QRS_NEXT_CUT()
PTP {E1 28976.886,E2 28976.886}
PTP {X 0,Y 607.919,A -85,B 0,C 180,E1 28976.886,E2 28976.886,E3 0,E4 0,E5 0,E6 0}
QRS_SPEED_INIT()
LIN {X 0,Y 607.919,Z 855,A -85,B 0,C 180,E1 28976.886,E2 28976.886,E3 0,E4 0,E5 0,E6 0} C_VEL
LIN {X 0,Y 607.919,Z 792.512,A -85,B 0,C 180,E1 28976.886,E2 28976.886} C_VEL
LIN {X 0,Y 607.919,Z 784.1,A -85,B 0,C 180,E1 28976.886,E2 28976.886} C_VEL
LIN {X 0,Y 607.91,Z 782.124,A -85,B 0,C 180,E1 28976.726,E2 28976.726} C_VEL
LIN {X 0,Y 607.918,Z 778.216,A -85,B 0,C 180,E1 28974.999,E2 28974.999} C_VEL
LIN {X 0,Y 607.918,Z 772.634,A -85,B 0,C 180,E1 28973.294,E2 28973.294} C_VEL
LIN {X 0,Y 607.917,Z 765.18,A -85,B 0,C 180,E1 28971.583,E2 28971.583} C_VEL
LIN {X 0,Y 607.91,Z 756.203,A -85,B 0,C 180,E1 28969.959,E2 28969.959} C_VEL
LIN {X 0,Y 607.915,Z 745.767,A -85,B 0,C 180,E1 28968.424,E2 28968.424} C_VEL
LIN {X 0,Y 607.915,Z 733.893,A -85,B 0,C 180,E1 28966.978,E2 28966.978} C_VEL
LIN {X 0,Y 607.913,Z 720.544,A -85,B 0,C 180,E1 28965.62,E2 28965.62} C_VEL
LIN {X 0,Y 607.917,Z 705.535,A -85,B 0,C 180,E1 28964.351,E2 28964.351} C_VEL
LIN {X 0,Y 607.92,Z 689.426,A -85,B 0,C 180,E1 28963.228,E2 28963.228} C_VEL
LIN {X 0,Y 607.911,Z 672.944,A -85,B 0,C 180,E1 28962.285,E2 28962.285} C_VEL
LIN {X 0,Y 607.914,Z 655.674,A -85,B 0,C 180,E1 28961.492,E2 28961.492} C_VEL
LIN {X 0,Y 607.918,Z 638.216,A -85,B 0,C 180,E1 28960.87,E2 28960.87} C_VEL
LIN {X 0,Y 607.911,Z 619.855,A -85,B 0,C 180,E1 28960.395,E2 28960.395} C_VEL
LIN {X 0,Y 607.907,Z 600.729,A -85,B 0,C 180,E1 28960.082,E2 28960.082} C_VEL
LIN {X 0,Y 607.893,Z 403.798,A -85,B 0,C 180,E1 28957.622,E2 28957.622} C_VEL
LIN {X 0,Y 607.907,Z 366.363,A -85,B 0,C 180,E1 28954.552,E2 28954.552} C_VEL
LIN {X 0,Y 607.851,Z 351.079,A -85,B 0,C 180,E1 28953.244,E2 28953.244} C_VEL
LIN {X 0,Y 607.85,Z 351.077,A -85,B 0,C 180,E1 28949.996,E2 28949.996} C_VEL
LIN {X 0,Y 607.849,Z 351.076,A -85,B 0,C 180,E1 28947.199,E2 28947.199} C_VEL
LIN {X 0,Y 607.849,Z 351.077,A -85,B 0,C 180,E1 28943.922,E2 28943.922} C_VEL
LIN {X 0,Y 607.845,Z 351.076,A -85,B 0,C 180,E1 28941.192,E2 28941.192} C_VEL
LIN {X 0,Y 607.851,Z 351.077,A -85,B 0,C 180,E1 28937.89,E2 28937.89} C_VEL
LIN {X 0,Y 607.845,Z 351.076,A -85,B 0,C 180,E1 28935.116,E2 28935.116} C_VEL
LIN {X 0,Y 607.851,Z 351.077,A -85,B 0,C 180,E1 28931.828,E2 28931.828} C_VEL
LIN {X 0,Y 607.845,Z 351.076,A -85,B 0,C 180,E1 28929.051,E2 28929.051} C_VEL
LIN {X 0,Y 607.848,Z 351.077,A -85,B 0,C 180,E1 28925.729,E2 28925.729} C_VEL
LIN {X 0,Y 607.845,Z 351.076,A -85,B 0,C 180,E1 28922.974,E2 28922.974} C_VEL
LIN {X 0,Y 607.848,Z 351.077,A -85,B 0,C 180,E1 28919.678,E2 28919.678} C_VEL
LIN {X 0,Y 607.845,Z 351.076,A -85,B 0,C 180,E1 28916.895,E2 28916.895} C_VEL
LIN {X 0,Y 607.845,Z 351.077,A -85,B 0,C 180,E1 28913.561,E2 28913.561} C_VEL
LIN {X 0,Y 607.847,Z 351.076,A -85,B 0,C 180,E1 28910.812,E2 28910.812} C_VEL
LIN {X 0,Y 607.846,Z 351.077,A -85,B 0,C 180,E1 28907.519,E2 28907.519} C_VEL
LIN {X 0,Y 607.843,Z 351.076,A -85,B 0,C 180,E1 28904.772,E2 28904.772} C_VEL
LIN {X 0,Y 607.848,Z 351.077,A -85,B 0,C 180,E1 28901.481,E2 28901.481} C_VEL
LIN {X 0,Y 607.845,Z 351.076,A -85,B 0,C 180,E1 28898.704,E2 28898.704} C_VEL
LIN {X 0,Y 607.845,Z 351.077,A -85,B 0,C 180,E1 28895.38,E2 28895.38} C_VEL
LIN {X 0,Y 607.844,Z 351.076,A -85,B 0,C 180,E1 28892.64,E2 28892.64} C_VEL
LIN {X 0,Y 607.847,Z 351.077,A -85,B 0,C 180,E1 28889.34,E2 28889.34} C_VEL
LIN {X 0,Y 607.848,Z 351.076,A -85,B 0,C 180,E1 28886.511,E2 28886.511} C_VEL
LIN {X 0,Y 607.848,Z 351.077,A -85,B 0,C 180,E1 28883.293,E2 28883.293} C_VEL
LIN {X 0,Y 607.842,Z 351.076,A -85,B 0,C 180,E1 28880.532,E2 28880.532} C_VEL
LIN {X 0,Y 607.85,Z 351.077,A -85,B 0,C 180,E1 28877.266,E2 28877.266} C_VEL
LIN {X 0,Y 607.837,Z 351.076,A -85,B 0,C 180,E1 28874.545,E2 28874.545} C_VEL
LIN {X 0,Y 607.864,Z 351.077,A -85,B 0,C 180,E1 28871.343,E2 28871.343} C_VEL
LIN {X 0,Y 607.833,Z 351.077,A -85,B 0,C 180,E1 28868.581,E2 28868.581} C_VEL
LIN {X 0,Y 607.885,Z 351.077,A -85,B 0,C 180,E1 28865.448,E2 28865.448} C_VEL
LIN {X 0,Y 607.832,Z 351.077,A -85,B 0,C 180,E1 28862.575,E2 28862.575} C_VEL
LIN {X 0,Y 607.906,Z 351.077,A -85,B 0,C 180,E1 28859.526,E2 28859.526} C_VEL
LIN {X 0,Y 607.83,Z 351.077,A -85,B 0,C 180,E1 28856.56,E2 28856.56} C_VEL
LIN {X 0,Y 607.913,Z 351.078,A -85,B 0,C 180,E1 28853.541,E2 28853.541} C_VEL
LIN {X 0,Y 607.83,Z 351.077,A -85,B 0,C 180,E1 28850.583,E2 28850.583} C_VEL
LIN {X 0,Y 607.903,Z 351.077,A -85,B 0,C 180,E1 28847.596,E2 28847.596} C_VEL
LIN {X 0,Y 607.831,Z 351.077,A -85,B 0,C 180,E1 28844.58,E2 28844.58} C_VEL
LIN {X 0,Y 607.883,Z 351.077,A -85,B 0,C 180,E1 28841.69,E2 28841.69} C_VEL
LIN {X 0,Y 607.832,Z 351.077,A -85,B 0,C 180,E1 28838.568,E2 28838.568} C_VEL
LIN {X 0,Y 607.859,Z 351.077,A -85,B 0,C 180,E1 28835.813,E2 28835.813} C_VEL
LIN {X 0,Y 607.837,Z 351.077,A -85,B 0,C 180,E1 28832.625,E2 28832.625} C_VEL
LIN {X 0,Y 607.855,Z 351.077,A -85,B 0,C 180,E1 28829.786,E2 28829.786} C_VEL
LIN {X 0,Y 607.837,Z 351.08,A -85,B 0,C 180,E1 28826.579,E2 28826.579} C_VEL
LIN {X 0,Y 607.829,Z 351.304,A -85,B 0,C 180,E1 28826.333,E2 28826.333} C_VEL
LIN {X 0,Y 607.917,Z 379.245,A -85,B 0,C 180,E1 28823.352,E2 28823.352} C_VEL
LIN {X 0,Y 607.876,Z 408.984,A -85,B 0,C 180,E1 28820.258,E2 28820.258} C_VEL
LIN {X 0,Y 607.915,Z 440.675,A -85,B 0,C 180,E1 28817.024,E2 28817.024} C_VEL
LIN {X 0,Y 607.889,Z 472.368,A -85,B 0,C 180,E1 28813.847,E2 28813.847} C_VEL
LIN {X 0,Y 607.915,Z 480.891,A -85,B 0,C 180,E1 28813.01,E2 28813.01} C_VEL
LIN {X 0,Y 607.868,Z 591.977,A -85,B 0,C 180,E1 28811.673,E2 28811.673} C_VEL
LIN {X 0,Y 607.896,Z 607.193,A -85,B 0,C 180,E1 28811.312,E2 28811.312} C_VEL
LIN {X 0,Y 607.914,Z 622.026,A -85,B 0,C 180,E1 28810.759,E2 28810.759} C_VEL
LIN {X 0,Y 607.88,Z 635.112,A -85,B 0,C 180,E1 28810.089,E2 28810.089} C_VEL
LIN {X 0,Y 607.918,Z 647.311,A -85,B 0,C 180,E1 28809.276,E2 28809.276} C_VEL
LIN {X 0,Y 607.919,Z 658.998,A -85,B 0,C 180,E1 28808.274,E2 28808.274} C_VEL
LIN {X 0,Y 607.918,Z 668.983,A -85,B 0,C 180,E1 28807.181,E2 28807.181} C_VEL
LIN {X 0,Y 607.917,Z 677.168,A -85,B 0,C 180,E1 28806.042,E2 28806.042} C_VEL
LIN {X 0,Y 607.918,Z 684.395,A -85,B 0,C 180,E1 28804.717,E2 28804.717} C_VEL
LIN {X 0,Y 607.917,Z 689.553,A -85,B 0,C 180,E1 28803.395,E2 28803.395} C_VEL
LIN {X 0,Y 607.916,Z 692.97,A -85,B 0,C 180,E1 28802.074,E2 28802.074} C_VEL
LIN {X 0,Y 607.918,Z 694.754,A -85,B 0,C 180,E1 28800.66,E2 28800.66} C_VEL
LIN {X 0,Y 607.914,Z 694.751,A -85,B 0,C 180,E1 28799.246,E2 28799.246} C_VEL
LIN {X 0,Y 607.919,Z 692.961,A -85,B 0,C 180,E1 28797.832,E2 28797.832} C_VEL
LIN {X 0,Y 607.919,Z 689.239,A -85,B 0,C 180,E1 28796.417,E2 28796.417} C_VEL
LIN {X 0,Y 607.916,Z 683.914,A -85,B 0,C 180,E1 28795.094,E2 28795.094} C_VEL
LIN {X 0,Y 607.918,Z 677.14,A -85,B 0,C 180,E1 28793.863,E2 28793.863} C_VEL
LIN {X 0,Y 607.917,Z 668.32,A -85,B 0,C 180,E1 28792.648,E2 28792.648} C_VEL
LIN {X 0,Y 607.918,Z 658.44,A -85,B 0,C 180,E1 28791.583,E2 28791.583} C_VEL
LIN {X 0,Y 607.92,Z 647.242,A -85,B 0,C 180,E1 28790.629,E2 28790.629} C_VEL
LIN {X 0,Y 607.891,Z 634.216,A -85,B 0,C 180,E1 28789.768,E2 28789.768} C_VEL
LIN {X 0,Y 607.917,Z 620.772,A -85,B 0,C 180,E1 28789.097,E2 28789.097} C_VEL
LIN {X 0,Y 607.912,Z 606.579,A -85,B 0,C 180,E1 28788.581,E2 28788.581} C_VEL
LIN {X 0,Y 607.912,Z 590.99,A -85,B 0,C 180,E1 28788.22,E2 28788.22} C_VEL
LIN {X 0,Y 607.918,Z 480.591,A -85,B 0,C 180,E1 28786.881,E2 28786.881} C_VEL
LIN {X 0,Y 607.909,Z 447.91,A -85,B 0,C 180,E1 28783.616,E2 28783.616} C_VEL
LIN {X 0,Y 607.91,Z 416.898,A -85,B 0,C 180,E1 28780.467,E2 28780.467} C_VEL
LIN {X 0,Y 607.864,Z 387.42,A -85,B 0,C 180,E1 28777.414,E2 28777.414} C_VEL
LIN {X 0,Y 607.87,Z 358.389,A -85,B 0,C 180,E1 28774.341,E2 28774.341} C_VEL
LIN {X 0,Y 607.832,Z 351.08,A -85,B 0,C 180,E1 28773.527,E2 28773.527} C_VEL
LIN {X 0,Y 607.89,Z 351.078,A -85,B 0,C 180,E1 28770.433,E2 28770.433} C_VEL
LIN {X 0,Y 607.831,Z 351.077,A -85,B 0,C 180,E1 28767.551,E2 28767.551} C_VEL
LIN {X 0,Y 607.904,Z 351.079,A -85,B 0,C 180,E1 28764.505,E2 28764.505} C_VEL
LIN {X 0,Y 607.831,Z 351.077,A -85,B 0,C 180,E1 28761.537,E2 28761.537} C_VEL
LIN {X 0,Y 607.911,Z 351.076,A -85,B 0,C 180,E1 28758.591,E2 28758.591} C_VEL
LIN {X 0,Y 607.832,Z 351.077,A -85,B 0,C 180,E1 28755.513,E2 28755.513} C_VEL
LIN {X 0,Y 607.909,Z 351.076,A -85,B 0,C 180,E1 28752.532,E2 28752.532} C_VEL
LIN {X 0,Y 607.834,Z 351.077,A -85,B 0,C 180,E1 28749.513,E2 28749.513} C_VEL
LIN {X 0,Y 607.897,Z 351.076,A -85,B 0,C 180,E1 28746.542,E2 28746.542} C_VEL
LIN {X 0,Y 607.836,Z 351.077,A -85,B 0,C 180,E1 28743.489,E2 28743.489} C_VEL
LIN {X 0,Y 607.897,Z 351.076,A -85,B 0,C 180,E1 28740.473,E2 28740.473} C_VEL
LIN {X 0,Y 607.854,Z 351.322,A -85,B 0,C 180,E1 28739.75,E2 28739.75} C_VEL
LIN {X 0,Y 607.905,Z 393.33,A -85,B 0,C 180,E1 28736.892,E2 28736.892} C_VEL
LIN {X 0,Y 607.901,Z 440.588,A -85,B 0,C 180,E1 28733.764,E2 28733.764} C_VEL
LIN {X 0,Y 607.913,Z 462.654,A -85,B 0,C 180,E1 28732.33,E2 28732.33} C_VEL
LIN {X 0,Y 607.916,Z 672.314,A -85,B 0,C 180,E1 28729.705,E2 28729.705} C_VEL
LIN {X 0,Y 607.917,Z 690.589,A -85,B 0,C 180,E1 28729.305,E2 28729.305} C_VEL
LIN {X 0,Y 607.913,Z 708.763,A -85,B 0,C 180,E1 28728.732,E2 28728.732} C_VEL
LIN {X 0,Y 607.914,Z 726.043,A -85,B 0,C 180,E1 28728.012,E2 28728.012} C_VEL
LIN {X 0,Y 607.919,Z 742.974,A -85,B 0,C 180,E1 28727.122,E2 28727.122} C_VEL
LIN {X 0,Y 607.916,Z 759.642,A -85,B 0,C 180,E1 28726.041,E2 28726.041} C_VEL
LIN {X 0,Y 607.917,Z 774.562,A -85,B 0,C 180,E1 28724.867,E2 28724.867} C_VEL
LIN {X 0,Y 607.918,Z 788.217,A -85,B 0,C 180,E1 28723.583,E2 28723.583} C_VEL
LIN {X 0,Y 607.916,Z 800.906,A -85,B 0,C 180,E1 28722.153,E2 28722.153} C_VEL
LIN {X 0,Y 607.91,Z 812.224,A -85,B 0,C 180,E1 28720.615,E2 28720.615} C_VEL
LIN {X 0,Y 607.919,Z 821.989,A -85,B 0,C 180,E1 28718.989,E2 28718.989} C_VEL
LIN {X 0,Y 607.915,Z 829.847,A -85,B 0,C 180,E1 28717.353,E2 28717.353} C_VEL
LIN {X 0,Y 607.907,Z 836.108,A -85,B 0,C 180,E1 28715.664,E2 28715.664} C_VEL
LIN {X 0,Y 607.917,Z 840.872,A -85,B 0,C 180,E1 28713.867,E2 28713.867} C_VEL
LIN {X 0,Y 607.911,Z 843.787,A -85,B 0,C 180,E1 28712.074,E2 28712.074} C_VEL
LIN {X 0,Y 607.907,Z 844.94,A -85,B 0,C 180,E1 28710.283,E2 28710.283} C_VEL
LIN {X 0,Y 607.916,Z 844.348,A -85,B 0,C 180,E1 28708.492,E2 28708.492} C_VEL
LIN {X 0,Y 607.908,Z 842.005,A -85,B 0,C 180,E1 28706.7,E2 28706.7} C_VEL
LIN {X 0,Y 607.917,Z 838.096,A -85,B 0,C 180,E1 28704.999,E2 28704.999} C_VEL
LIN {X 0,Y 607.912,Z 832.467,A -85,B 0,C 180,E1 28703.294,E2 28703.294} C_VEL
LIN {X 0,Y 607.914,Z 825.422,A -85,B 0,C 180,E1 28701.678,E2 28701.678} C_VEL
LIN {X 0,Y 607.91,Z 816.508,A -85,B 0,C 180,E1 28700.055,E2 28700.055} C_VEL
LIN {X 0,Y 607.919,Z 806.143,A -85,B 0,C 180,E1 28698.521,E2 28698.521} C_VEL
LIN {X 0,Y 607.912,Z 794.344,A -85,B 0,C 180,E1 28697.074,E2 28697.074} C_VEL
LIN {X 0,Y 607.916,Z 781.087,A -85,B 0,C 180,E1 28695.717,E2 28695.717} C_VEL
LIN {X 0,Y 607.915,Z 766.232,A -85,B 0,C 180,E1 28694.449,E2 28694.449} C_VEL
LIN {X 0,Y 607.917,Z 750.215,A -85,B 0,C 180,E1 28693.321,E2 28693.321} C_VEL
LIN {X 0,Y 607.911,Z 734.022,A -85,B 0,C 180,E1 28692.384,E2 28692.384} C_VEL
LIN {X 0,Y 607.913,Z 717.059,A -85,B 0,C 180,E1 28691.591,E2 28691.591} C_VEL
LIN {X 0,Y 607.914,Z 699.218,A -85,B 0,C 180,E1 28690.945,E2 28690.945} C_VEL
LIN {X 0,Y 607.914,Z 680.196,A -85,B 0,C 180,E1 28690.447,E2 28690.447} C_VEL
LIN {X 0,Y 607.915,Z 660.799,A -85,B 0,C 180,E1 28690.128,E2 28690.128} C_VEL
LIN {X 0,Y 607.912,Z 462.258,A -85,B 0,C 180,E1 28687.645,E2 28687.645} C_VEL
LIN {X 0,Y 607.897,Z 415.384,A -85,B 0,C 180,E1 28684.577,E2 28684.577} C_VEL
LIN {X 0,Y 607.899,Z 370.488,A -85,B 0,C 180,E1 28681.565,E2 28681.565} C_VEL
LIN {X 0,Y 607.857,Z 351.08,A -85,B 0,C 180,E1 28680.214,E2 28680.214} C_VEL
LIN {X 0,Y 607.844,Z 351.076,A -85,B 0,C 180,E1 28677.011,E2 28677.011} C_VEL
LIN {X 0,Y 607.846,Z 351.077,A -85,B 0,C 180,E1 28674.271,E2 28674.271} C_VEL
LIN {X 0,Y 607.844,Z 351.076,A -85,B 0,C 180,E1 28670.949,E2 28670.949} C_VEL
LIN {X 0,Y 607.844,Z 351.077,A -85,B 0,C 180,E1 28668.226,E2 28668.226} C_VEL
LIN {X 0,Y 607.842,Z 351.077,A -85,B 0,C 180,E1 28664.884,E2 28664.884} C_VEL
LIN {X 0,Y 607.846,Z 351.077,A -85,B 0,C 180,E1 28662.109,E2 28662.109} C_VEL
LIN {X 0,Y 607.842,Z 351.077,A -85,B 0,C 180,E1 28658.808,E2 28658.808} C_VEL
LIN {X 0,Y 607.841,Z 351.077,A -85,B 0,C 180,E1 28656.078,E2 28656.078} C_VEL
LIN {X 0,Y 607.843,Z 351.077,A -85,B 0,C 180,E1 28652.764,E2 28652.764} C_VEL
LIN {X 0,Y 607.84,Z 351.078,A -85,B 0,C 180,E1 28650.004,E2 28650.004} C_VEL
LIN {X 0,Y 607.839,Z 351.079,A -85,B 0,C 180,E1 28646.657,E2 28646.657} C_VEL
LIN {X 0,Y 607.904,Z 381.923,A -85,B 0,C 180,E1 28644.073,E2 28644.073} C_VEL
LIN {X 0,Y 607.893,Z 404.166,A -85,B 0,C 180,E1 28642.267,E2 28642.267} C_VEL
LIN {X 0,Y 607.915,Z 611.934,A -85,B 0,C 180,E1 28639.667,E2 28639.667} C_VEL
LIN {X 0,Y 607.915,Z 630.91,A -85,B 0,C 180,E1 28639.251,E2 28639.251} C_VEL
LIN {X 0,Y 607.913,Z 649.193,A -85,B 0,C 180,E1 28638.67,E2 28638.67} C_VEL
LIN {X 0,Y 607.917,Z 667.162,A -85,B 0,C 180,E1 28637.912,E2 28637.912} C_VEL
LIN {X 0,Y 607.919,Z 683.868,A -85,B 0,C 180,E1 28637.023,E2 28637.023} C_VEL
LIN {X 0,Y 607.917,Z 699.702,A -85,B 0,C 180,E1 28635.991,E2 28635.991} C_VEL
LIN {X 0,Y 607.915,Z 714.603,A -85,B 0,C 180,E1 28634.818,E2 28634.818} C_VEL
LIN {X 0,Y 607.917,Z 728.521,A -85,B 0,C 180,E1 28633.506,E2 28633.506} C_VEL
LIN {X 0,Y 607.916,Z 741.322,A -85,B 0,C 180,E1 28632.057,E2 28632.057} C_VEL
LIN {X 0,Y 607.91,Z 752.564,A -85,B 0,C 180,E1 28630.519,E2 28630.519} C_VEL
LIN {X 0,Y 607.914,Z 762.265,A -85,B 0,C 180,E1 28628.894,E2 28628.894} C_VEL
LIN {X 0,Y 607.915,Z 769.988,A -85,B 0,C 180,E1 28627.276,E2 28627.276} C_VEL
LIN {X 0,Y 607.917,Z 776.266,A -85,B 0,C 180,E1 28625.569,E2 28625.569} C_VEL
LIN {X 0,Y 607.918,Z 780.98,A -85,B 0,C 180,E1 28623.772,E2 28623.772} C_VEL
LIN {X 0,Y 607.908,Z 783.846,A -85,B 0,C 180,E1 28621.979,E2 28621.979} C_VEL
LIN {X 0,Y 607.908,Z 784.951,A -85,B 0,C 180,E1 28620.188,E2 28620.188} C_VEL
LIN {X 0,Y 607.914,Z 784.313,A -85,B 0,C 180,E1 28618.398,E2 28618.398} C_VEL
LIN {X 0,Y 607.91,Z 782.124,A -85,B 0,C 180,E1 28616.726,E2 28616.726} C_VEL
LIN {X 0,Y 606.898,Z 780.802,A -85,B 0,C 180,E1 28616.011,E2 28616.011} C_VEL
LIN {X 0,Y 602.275,Z 777.568,A -85,B 0,C 180,E1 28614.68,E2 28614.68} C_VEL
LIN {X 0,Y 600.12,Z 774.916,A -85,B 0,C 180,E1 28613.834,E2 28613.834} C_VEL
LIN {X 0,Y 599.921,Z 773.838,A -85,B 0,C 180,E1 28613.532,E2 28613.532} C_VEL
LIN {X 0,Y 599.923,Z 767.023,A -85,B 0,C 180,E1 28611.856,E2 28611.856} C_VEL
LIN {X 0,Y 599.942,Z 758.507,A -85,B 0,C 180,E1 28610.212,E2 28610.212} C_VEL
LIN {X 0,Y 599.964,Z 748.584,A -85,B 0,C 180,E1 28608.659,E2 28608.659} C_VEL
LIN {X 0,Y 600.001,Z 737.285,A -85,B 0,C 180,E1 28607.195,E2 28607.195} C_VEL
LIN {X 0,Y 600.041,Z 724.079,A -85,B 0,C 180,E1 28605.772,E2 28605.772} C_VEL
LIN {X 0,Y 600.088,Z 709.205,A -85,B 0,C 180,E1 28604.439,E2 28604.439} C_VEL
LIN {X 0,Y 600.143,Z 693.862,A -85,B 0,C 180,E1 28603.298,E2 28603.298} C_VEL
LIN {X 0,Y 600.196,Z 677.652,A -85,B 0,C 180,E1 28602.305,E2 28602.305} C_VEL
LIN {X 0,Y 600.252,Z 660.363,A -85,B 0,C 180,E1 28601.448,E2 28601.448} C_VEL
LIN {X 0,Y 600.311,Z 642.895,A -85,B 0,C 180,E1 28600.773,E2 28600.773} C_VEL
LIN {X 0,Y 600.35,Z 624.369,A -85,B 0,C 180,E1 28600.243,E2 28600.243} C_VEL
LIN {X 0,Y 600.381,Z 605.347,A -85,B 0,C 180,E1 28599.885,E2 28599.885} C_VEL
LIN {X 0,Y 600.353,Z 404.565,A -85,B 0,C 180,E1 28597.353,E2 28597.353} C_VEL
LIN {X 0,Y 600.289,Z 400.607,A -85,B 0,C 180,E1 28597.06,E2 28597.06} C_VEL
LIN {X 0,Y 600.342,Z 363.521,A -85,B 0,C 180,E1 28593.969,E2 28593.969} C_VEL
LIN {X 0,Y 600.208,Z 353.401,A -85,B 0,C 180,E1 28593.104,E2 28593.104} C_VEL
LIN {X 0,Y 599.94,Z 352.069,A -85,B 0,C 180,E1 28592.963,E2 28592.963} C_VEL
LIN {X 0,Y 599.901,Z 352.066,A -85,B 0,C 180,E1 28589.778,E2 28589.778} C_VEL
LIN {X 0,Y 599.942,Z 352.065,A -85,B 0,C 180,E1 28586.863,E2 28586.863} C_VEL
LIN {X 0,Y 599.9,Z 352.066,A -85,B 0,C 180,E1 28583.723,E2 28583.723} C_VEL
LIN {X 0,Y 599.944,Z 352.065,A -85,B 0,C 180,E1 28580.802,E2 28580.802} C_VEL
LIN {X 0,Y 599.9,Z 352.066,A -85,B 0,C 180,E1 28577.674,E2 28577.674} C_VEL
LIN {X 0,Y 599.938,Z 352.065,A -85,B 0,C 180,E1 28574.767,E2 28574.767} C_VEL
LIN {X 0,Y 599.903,Z 352.066,A -85,B 0,C 180,E1 28571.684,E2 28571.684} C_VEL
LIN {X 0,Y 599.918,Z 352.065,A -85,B 0,C 180,E1 28568.892,E2 28568.892} C_VEL
LIN {X 0,Y 599.907,Z 352.066,A -85,B 0,C 180,E1 28565.686,E2 28565.686} C_VEL
LIN {X 0,Y 599.915,Z 352.065,A -85,B 0,C 180,E1 28562.859,E2 28562.859} C_VEL
LIN {X 0,Y 599.909,Z 352.066,A -85,B 0,C 180,E1 28559.67,E2 28559.67} C_VEL
LIN {X 0,Y 599.909,Z 352.065,A -85,B 0,C 180,E1 28556.851,E2 28556.851} C_VEL
LIN {X 0,Y 599.906,Z 352.066,A -85,B 0,C 180,E1 28553.554,E2 28553.554} C_VEL
LIN {X 0,Y 599.911,Z 352.065,A -85,B 0,C 180,E1 28550.77,E2 28550.77} C_VEL
LIN {X 0,Y 599.904,Z 352.065,A -85,B 0,C 180,E1 28547.458,E2 28547.458} C_VEL
LIN {X 0,Y 599.911,Z 352.065,A -85,B 0,C 180,E1 28544.675,E2 28544.675} C_VEL
LIN {X 0,Y 599.907,Z 352.066,A -85,B 0,C 180,E1 28541.44,E2 28541.44} C_VEL
LIN {X 0,Y 599.911,Z 352.065,A -85,B 0,C 180,E1 28538.627,E2 28538.627} C_VEL
LIN {X 0,Y 599.905,Z 352.066,A -85,B 0,C 180,E1 28535.356,E2 28535.356} C_VEL
LIN {X 0,Y 599.91,Z 352.065,A -85,B 0,C 180,E1 28532.579,E2 28532.579} C_VEL
LIN {X 0,Y 599.907,Z 352.066,A -85,B 0,C 180,E1 28529.332,E2 28529.332} C_VEL
LIN {X 0,Y 599.913,Z 352.065,A -85,B 0,C 180,E1 28526.464,E2 28526.464} C_VEL
LIN {X 0,Y 599.903,Z 352.066,A -85,B 0,C 180,E1 28523.204,E2 28523.204} C_VEL
LIN {X 0,Y 599.912,Z 352.065,A -85,B 0,C 180,E1 28520.406,E2 28520.406} C_VEL
LIN {X 0,Y 599.905,Z 352.066,A -85,B 0,C 180,E1 28517.167,E2 28517.167} C_VEL
LIN {X 0,Y 599.905,Z 352.065,A -85,B 0,C 180,E1 28514.434,E2 28514.434} C_VEL
LIN {X 0,Y 599.906,Z 352.066,A -85,B 0,C 180,E1 28511.135,E2 28511.135} C_VEL
LIN {X 0,Y 599.903,Z 352.065,A -85,B 0,C 180,E1 28508.387,E2 28508.387} C_VEL
LIN {X 0,Y 599.905,Z 352.066,A -85,B 0,C 180,E1 28505.051,E2 28505.051} C_VEL
LIN {X 0,Y 599.908,Z 352.065,A -85,B 0,C 180,E1 28502.253,E2 28502.253} C_VEL
LIN {X 0,Y 599.902,Z 352.066,A -85,B 0,C 180,E1 28498.947,E2 28498.947} C_VEL
LIN {X 0,Y 599.914,Z 352.066,A -85,B 0,C 180,E1 28496.099,E2 28496.099} C_VEL
LIN {X 0,Y 599.902,Z 352.066,A -85,B 0,C 180,E1 28492.89,E2 28492.89} C_VEL
LIN {X 0,Y 599.901,Z 352.066,A -85,B 0,C 180,E1 28490.206,E2 28490.206} C_VEL
LIN {X 0,Y 599.906,Z 352.066,A -85,B 0,C 180,E1 28486.888,E2 28486.888} C_VEL
LIN {X 0,Y 599.9,Z 352.066,A -85,B 0,C 180,E1 28484.162,E2 28484.162} C_VEL
LIN {X 0,Y 599.914,Z 352.066,A -85,B 0,C 180,E1 28480.92,E2 28480.92} C_VEL
LIN {X 0,Y 599.894,Z 352.066,A -85,B 0,C 180,E1 28478.196,E2 28478.196} C_VEL
LIN {X 0,Y 599.938,Z 352.067,A -85,B 0,C 180,E1 28475.084,E2 28475.084} C_VEL
LIN {X 0,Y 599.895,Z 352.066,A -85,B 0,C 180,E1 28472.145,E2 28472.145} C_VEL
LIN {X 0,Y 599.938,Z 352.067,A -85,B 0,C 180,E1 28469.011,E2 28469.011} C_VEL
LIN {X 0,Y 599.917,Z 352.195,A -85,B 0,C 180,E1 28466.61,E2 28466.61} C_VEL
LIN {X 0,Y 600.229,Z 357.801,A -85,B 0,C 180,E1 28465.983,E2 28465.983} C_VEL
LIN {X 0,Y 600.159,Z 387.539,A -85,B 0,C 180,E1 28462.789,E2 28462.789} C_VEL
LIN {X 0,Y 600.14,Z 416.304,A -85,B 0,C 180,E1 28459.768,E2 28459.768} C_VEL
LIN {X 0,Y 600.069,Z 448.014,A -85,B 0,C 180,E1 28456.503,E2 28456.503} C_VEL
LIN {X 0,Y 600.02,Z 480.175,A -85,B 0,C 180,E1 28453.246,E2 28453.246} C_VEL
LIN {X 0,Y 600.084,Z 481.335,A -85,B 0,C 180,E1 28453.178,E2 28453.178} C_VEL
LIN {X 0,Y 600.032,Z 592.357,A -85,B 0,C 180,E1 28451.821,E2 28451.821} C_VEL
LIN {X 0,Y 600.039,Z 607.13,A -85,B 0,C 180,E1 28451.464,E2 28451.464} C_VEL
LIN {X 0,Y 600.035,Z 620.903,A -85,B 0,C 180,E1 28450.951,E2 28450.951} C_VEL
LIN {X 0,Y 599.975,Z 634.324,A -85,B 0,C 180,E1 28450.272,E2 28450.272} C_VEL
LIN {X 0,Y 599.984,Z 647.304,A -85,B 0,C 180,E1 28449.399,E2 28449.399} C_VEL
LIN {X 0,Y 599.962,Z 659.004,A -85,B 0,C 180,E1 28448.385,E2 28448.385} C_VEL
LIN {X 0,Y 599.943,Z 668.988,A -85,B 0,C 180,E1 28447.277,E2 28447.277} C_VEL
LIN {X 0,Y 599.929,Z 677.171,A -85,B 0,C 180,E1 28446.123,E2 28446.123} C_VEL
LIN {X 0,Y 599.923,Z 684.401,A -85,B 0,C 180,E1 28444.78,E2 28444.78} C_VEL
LIN {X 0,Y 599.918,Z 689.551,A -85,B 0,C 180,E1 28443.44,E2 28443.44} C_VEL
LIN {X 0,Y 599.917,Z 692.97,A -85,B 0,C 180,E1 28442.101,E2 28442.101} C_VEL
LIN {X 0,Y 599.918,Z 694.755,A -85,B 0,C 180,E1 28440.669,E2 28440.669} C_VEL
LIN {X 0,Y 599.914,Z 694.751,A -85,B 0,C 180,E1 28439.236,E2 28439.236} C_VEL
LIN {X 0,Y 599.918,Z 692.959,A -85,B 0,C 180,E1 28437.803,E2 28437.803} C_VEL
LIN {X 0,Y 599.92,Z 689.233,A -85,B 0,C 180,E1 28436.369,E2 28436.369} C_VEL
LIN {X 0,Y 599.922,Z 683.915,A -85,B 0,C 180,E1 28435.028,E2 28435.028} C_VEL
LIN {X 0,Y 599.93,Z 677.135,A -85,B 0,C 180,E1 28433.781,E2 28433.781} C_VEL
LIN {X 0,Y 599.942,Z 668.575,A -85,B 0,C 180,E1 28432.582,E2 28432.582} C_VEL
LIN {X 0,Y 599.962,Z 658.433,A -85,B 0,C 180,E1 28431.47,E2 28431.47} C_VEL
LIN {X 0,Y 599.986,Z 647.219,A -85,B 0,C 180,E1 28430.504,E2 28430.504} C_VEL
LIN {X 0,Y 599.985,Z 634.211,A -85,B 0,C 180,E1 28429.632,E2 28429.632} C_VEL
LIN {X 0,Y 600.037,Z 620.741,A -85,B 0,C 180,E1 28428.952,E2 28428.952} C_VEL
LIN {X 0,Y 600.056,Z 607.482,A -85,B 0,C 180,E1 28428.458,E2 28428.458} C_VEL
LIN {X 0,Y 600.076,Z 591.952,A -85,B 0,C 180,E1 28428.082,E2 28428.082} C_VEL
LIN {X 0,Y 600.019,Z 480.585,A -85,B 0,C 180,E1 28426.705,E2 28426.705} C_VEL
LIN {X 0,Y 600.063,Z 448.391,A -85,B 0,C 180,E1 28423.445,E2 28423.445} C_VEL
LIN {X 0,Y 600.135,Z 417.171,A -85,B 0,C 180,E1 28420.232,E2 28420.232} C_VEL
LIN {X 0,Y 600.165,Z 387.902,A -85,B 0,C 180,E1 28417.159,E2 28417.159} C_VEL
LIN {X 0,Y 600.226,Z 357.655,A -85,B 0,C 180,E1 28413.911,E2 28413.911} C_VEL
LIN {X 0,Y 599.906,Z 352.071,A -85,B 0,C 180,E1 28413.28,E2 28413.28} C_VEL
LIN {X 0,Y 599.904,Z 352.067,A -85,B 0,C 180,E1 28409.999,E2 28409.999} C_VEL
LIN {X 0,Y 599.907,Z 352.066,A -85,B 0,C 180,E1 28407.202,E2 28407.202} C_VEL
LIN {X 0,Y 599.905,Z 352.067,A -85,B 0,C 180,E1 28403.935,E2 28403.935} C_VEL
LIN {X 0,Y 599.91,Z 352.066,A -85,B 0,C 180,E1 28401.109,E2 28401.109} C_VEL
LIN {X 0,Y 599.903,Z 352.066,A -85,B 0,C 180,E1 28397.803,E2 28397.803} C_VEL
LIN {X 0,Y 599.916,Z 352.066,A -85,B 0,C 180,E1 28394.965,E2 28394.965} C_VEL
LIN {X 0,Y 599.908,Z 352.066,A -85,B 0,C 180,E1 28391.811,E2 28391.811} C_VEL
LIN {X 0,Y 599.906,Z 352.066,A -85,B 0,C 180,E1 28389.043,E2 28389.043} C_VEL
LIN {X 0,Y 599.905,Z 352.067,A -85,B 0,C 180,E1 28385.686,E2 28385.686} C_VEL
LIN {X 0,Y 599.915,Z 352.066,A -85,B 0,C 180,E1 28382.86,E2 28382.86} C_VEL
LIN {X 0,Y 599.966,Z 352.116,A -85,B 0,C 180,E1 28380.126,E2 28380.126} C_VEL
LIN {X 0,Y 600.577,Z 355.651,A -85,B 0,C 180,E1 28379.845,E2 28379.845} C_VEL
LIN {X 0,Y 600.507,Z 397.267,A -85,B 0,C 180,E1 28376.983,E2 28376.983} C_VEL
LIN {X 0,Y 600.374,Z 443.739,A -85,B 0,C 180,E1 28373.872,E2 28373.872} C_VEL
LIN {X 0,Y 600.419,Z 463.183,A -85,B 0,C 180,E1 28372.617,E2 28372.617} C_VEL
LIN {X 0,Y 600.375,Z 672.313,A -85,B 0,C 180,E1 28369.963,E2 28369.963} C_VEL
LIN {X 0,Y 600.337,Z 691.273,A -85,B 0,C 180,E1 28369.538,E2 28369.538} C_VEL
LIN {X 0,Y 600.285,Z 709.404,A -85,B 0,C 180,E1 28368.954,E2 28368.954} C_VEL
LIN {X 0,Y 600.231,Z 727.054,A -85,B 0,C 180,E1 28368.2,E2 28368.2} C_VEL
LIN {X 0,Y 600.179,Z 743.704,A -85,B 0,C 180,E1 28367.305,E2 28367.305} C_VEL
LIN {X 0,Y 600.122,Z 759.639,A -85,B 0,C 180,E1 28366.255,E2 28366.255} C_VEL
LIN {X 0,Y 600.069,Z 774.563,A -85,B 0,C 180,E1 28365.066,E2 28365.066} C_VEL
LIN {X 0,Y 600.02,Z 788.019,A -85,B 0,C 180,E1 28363.786,E2 28363.786} C_VEL
LIN {X 0,Y 599.982,Z 800.907,A -85,B 0,C 180,E1 28362.316,E2 28362.316} C_VEL
LIN {X 0,Y 599.953,Z 812.225,A -85,B 0,C 180,E1 28360.758,E2 28360.758} C_VEL
LIN {X 0,Y 599.939,Z 821.99,A -85,B 0,C 180,E1 28359.11,E2 28359.11} C_VEL
LIN {X 0,Y 599.925,Z 830.027,A -85,B 0,C 180,E1 28357.409,E2 28357.409} C_VEL
LIN {X 0,Y 599.911,Z 836.41,A -85,B 0,C 180,E1 28355.643,E2 28355.643} C_VEL
LIN {X 0,Y 599.917,Z 840.873,A -85,B 0,C 180,E1 28353.918,E2 28353.918} C_VEL
LIN {X 0,Y 599.911,Z 843.788,A -85,B 0,C 180,E1 28352.101,E2 28352.101} C_VEL
LIN {X 0,Y 599.907,Z 844.94,A -85,B 0,C 180,E1 28350.286,E2 28350.286} C_VEL
LIN {X 0,Y 599.915,Z 844.348,A -85,B 0,C 180,E1 28348.472,E2 28348.472} C_VEL
LIN {X 0,Y 599.907,Z 842.005,A -85,B 0,C 180,E1 28346.656,E2 28346.656} C_VEL
LIN {X 0,Y 599.919,Z 838.096,A -85,B 0,C 180,E1 28344.932,E2 28344.932} C_VEL
LIN {X 0,Y 599.92,Z 832.467,A -85,B 0,C 180,E1 28343.204,E2 28343.204} C_VEL
LIN {X 0,Y 599.927,Z 825.423,A -85,B 0,C 180,E1 28341.566,E2 28341.566} C_VEL
LIN {X 0,Y 599.942,Z 816.509,A -85,B 0,C 180,E1 28339.922,E2 28339.922} C_VEL
LIN {X 0,Y 599.969,Z 806.145,A -85,B 0,C 180,E1 28338.367,E2 28338.367} C_VEL
LIN {X 0,Y 600.001,Z 794.345,A -85,B 0,C 180,E1 28336.901,E2 28336.901} C_VEL
LIN {X 0,Y 600.047,Z 780.76,A -85,B 0,C 180,E1 28335.494,E2 28335.494} C_VEL
LIN {X 0,Y 600.102,Z 766.231,A -85,B 0,C 180,E1 28334.241,E2 28334.241} C_VEL
LIN {X 0,Y 600.164,Z 750.218,A -85,B 0,C 180,E1 28333.099,E2 28333.099} C_VEL
LIN {X 0,Y 600.216,Z 733.031,A -85,B 0,C 180,E1 28332.101,E2 28332.101} C_VEL
LIN {X 0,Y 600.277,Z 715.679,A -85,B 0,C 180,E1 28331.294,E2 28331.294} C_VEL
LIN {X 0,Y 600.328,Z 697.644,A -85,B 0,C 180,E1 28330.648,E2 28330.648} C_VEL
LIN {X 0,Y 600.366,Z 679.132,A -85,B 0,C 180,E1 28330.17,E2 28330.17} C_VEL
LIN {X 0,Y 600.391,Z 659.39,A -85,B 0,C 180,E1 28329.851,E2 28329.851} C_VEL
LIN {X 0,Y 600.361,Z 462.791,A -85,B 0,C 180,E1 28327.376,E2 28327.376} C_VEL
LIN {X 0,Y 600.446,Z 416.959,A -85,B 0,C 180,E1 28324.345,E2 28324.345} C_VEL
LIN {X 0,Y 600.578,Z 372.064,A -85,B 0,C 180,E1 28321.295,E2 28321.295} C_VEL
LIN {X 0,Y 600.409,Z 353.948,A -85,B 0,C 180,E1 28320.027,E2 28320.027} C_VEL
LIN {X 0,Y 599.965,Z 352.064,A -85,B 0,C 180,E1 28319.843,E2 28319.843} C_VEL
LIN {X 0,Y 599.896,Z 352.066,A -85,B 0,C 180,E1 28316.746,E2 28316.746} C_VEL
LIN {X 0,Y 599.966,Z 352.067,A -85,B 0,C 180,E1 28313.728,E2 28313.728} C_VEL
LIN {X 0,Y 599.894,Z 352.066,A -85,B 0,C 180,E1 28310.657,E2 28310.657} C_VEL
LIN {X 0,Y 599.96,Z 352.068,A -85,B 0,C 180,E1 28307.679,E2 28307.679} C_VEL
LIN {X 0,Y 599.894,Z 352.066,A -85,B 0,C 180,E1 28304.627,E2 28304.627} C_VEL
LIN {X 0,Y 599.955,Z 352.067,A -85,B 0,C 180,E1 28301.679,E2 28301.679} C_VEL
LIN {X 0,Y 599.894,Z 352.066,A -85,B 0,C 180,E1 28298.584,E2 28298.584} C_VEL
LIN {X 0,Y 599.955,Z 352.067,A -85,B 0,C 180,E1 28295.582,E2 28295.582} C_VEL
LIN {X 0,Y 599.893,Z 352.067,A -85,B 0,C 180,E1 28292.502,E2 28292.502} C_VEL
LIN {X 0,Y 599.951,Z 352.068,A -85,B 0,C 180,E1 28289.547,E2 28289.547} C_VEL
LIN {X 0,Y 599.941,Z 352.201,A -85,B 0,C 180,E1 28286.921,E2 28286.921} C_VEL
LIN {X 0,Y 600.332,Z 356.094,A -85,B 0,C 180,E1 28286.571,E2 28286.571} C_VEL
LIN {X 0,Y 600.314,Z 391.001,A -85,B 0,C 180,E1 28283.643,E2 28283.643} C_VEL
LIN {X 0,Y 600.332,Z 404.43,A -85,B 0,C 180,E1 28282.56,E2 28282.56} C_VEL
LIN {X 0,Y 600.385,Z 596.679,A -85,B 0,C 180,E1 28280.138,E2 28280.138} C_VEL
LIN {X 0,Y 600.367,Z 617.841,A -85,B 0,C 180,E1 28279.81,E2 28279.81} C_VEL
LIN {X 0,Y 600.331,Z 636.441,A -85,B 0,C 180,E1 28279.343,E2 28279.343} C_VEL
LIN {X 0,Y 600.281,Z 654.591,A -85,B 0,C 180,E1 28278.704,E2 28278.704} C_VEL
LIN {X 0,Y 600.222,Z 672.155,A -85,B 0,C 180,E1 28277.899,E2 28277.899} C_VEL
LIN {X 0,Y 600.168,Z 688.701,A -85,B 0,C 180,E1 28276.95,E2 28276.95} C_VEL
LIN {X 0,Y 600.111,Z 704.847,A -85,B 0,C 180,E1 28275.819,E2 28275.819} C_VEL
LIN {X 0,Y 600.056,Z 719.573,A -85,B 0,C 180,E1 28274.573,E2 28274.573} C_VEL
LIN {X 0,Y 600.01,Z 733.111,A -85,B 0,C 180,E1 28273.197,E2 28273.197} C_VEL
LIN {X 0,Y 599.975,Z 745.113,A -85,B 0,C 180,E1 28271.731,E2 28271.731} C_VEL
LIN {X 0,Y 599.948,Z 755.669,A -85,B 0,C 180,E1 28270.175,E2 28270.175} C_VEL
LIN {X 0,Y 599.924,Z 764.754,A -85,B 0,C 180,E1 28268.53,E2 28268.53} C_VEL
LIN {X 0,Y 599.918,Z 772.305,A -85,B 0,C 180,E1 28266.796,E2 28266.796} C_VEL
LIN {X 0,Y 599.918,Z 777.978,A -85,B 0,C 180,E1 28265.068,E2 28265.068} C_VEL
LIN {X 0,Y 599.915,Z 782.006,A -85,B 0,C 180,E1 28263.301,E2 28263.301} C_VEL
LIN {X 0,Y 599.917,Z 784.32,A -85,B 0,C 180,E1 28261.528,E2 28261.528} C_VEL
LIN {X 0,Y 599.915,Z 784.95,A -85,B 0,C 180,E1 28259.713,E2 28259.713} C_VEL
LIN {X 0,Y 599.906,Z 783.844,A -85,B 0,C 180,E1 28257.899,E2 28257.899} C_VEL
LIN {X 0,Y 599.914,Z 780.971,A -85,B 0,C 180,E1 28256.082,E2 28256.082} C_VEL
LIN {X 0,Y 599.91,Z 776.248,A -85,B 0,C 180,E1 28254.261,E2 28254.261} C_VEL
LIN {X 0,Y 599.921,Z 773.838,A -85,B 0,C 180,E1 28253.532,E2 28253.532} C_VEL
LIN {X 0,Y 598.925,Z 771.317,A -85,B 0,C 180,E1 28252.84,E2 28252.84} C_VEL
LIN {X 0,Y 592.681,Z 763.557,A -85,B 0,C 180,E1 28251.03,E2 28251.03} C_VEL
LIN {X 0,Y 591.959,Z 760.581,A -85,B 0,C 180,E1 28250.452,E2 28250.452} C_VEL
LIN {X 0,Y 592.002,Z 751.224,A -85,B 0,C 180,E1 28248.897,E2 28248.897} C_VEL
LIN {X 0,Y 592.064,Z 739.717,A -85,B 0,C 180,E1 28247.318,E2 28247.318} C_VEL
LIN {X 0,Y 592.151,Z 726.572,A -85,B 0,C 180,E1 28245.828,E2 28245.828} C_VEL
LIN {X 0,Y 592.253,Z 712.217,A -85,B 0,C 180,E1 28244.479,E2 28244.479} C_VEL
LIN {X 0,Y 592.366,Z 696.767,A -85,B 0,C 180,E1 28243.274,E2 28243.274} C_VEL
LIN {X 0,Y 592.482,Z 680.229,A -85,B 0,C 180,E1 28242.215,E2 28242.215} C_VEL
LIN {X 0,Y 592.597,Z 662.601,A -85,B 0,C 180,E1 28241.302,E2 28241.302} C_VEL
LIN {X 0,Y 592.713,Z 644.154,A -85,B 0,C 180,E1 28240.561,E2 28240.561} C_VEL
LIN {X 0,Y 592.799,Z 625.14,A -85,B 0,C 180,E1 28239.999,E2 28239.999} C_VEL
LIN {X 0,Y 592.864,Z 605.805,A -85,B 0,C 180,E1 28239.626,E2 28239.626} C_VEL
LIN {X 0,Y 592.965,Z 405.725,A -85,B 0,C 180,E1 28237.07,E2 28237.07} C_VEL
LIN {X 0,Y 592.667,Z 403.772,A -85,B 0,C 180,E1 28237.014,E2 28237.014} C_VEL
LIN {X 0,Y 592.835,Z 366.656,A -85,B 0,C 180,E1 28233.883,E2 28233.883} C_VEL
LIN {X 0,Y 592.624,Z 355.341,A -85,B 0,C 180,E1 28232.9,E2 28232.9} C_VEL
LIN {X 0,Y 592.036,Z 353.055,A -85,B 0,C 180,E1 28232.654,E2 28232.654} C_VEL
LIN {X 0,Y 591.959,Z 353.056,A -85,B 0,C 180,E1 28229.554,E2 28229.554} C_VEL
LIN {X 0,Y 592.033,Z 353.055,A -85,B 0,C 180,E1 28226.478,E2 28226.478} C_VEL
LIN {X 0,Y 591.96,Z 353.055,A -85,B 0,C 180,E1 28223.399,E2 28223.399} C_VEL
LIN {X 0,Y 592.003,Z 353.055,A -85,B 0,C 180,E1 28220.2,E2 28220.2} C_VEL
LIN {X 0,Y 591.964,Z 353.054,A -85,B 0,C 180,E1 28217.234,E2 28217.234} C_VEL
LIN {X 0,Y 591.986,Z 353.055,A -85,B 0,C 180,E1 28213.986,E2 28213.986} C_VEL
LIN {X 0,Y 591.968,Z 353.054,A -85,B 0,C 180,E1 28211.075,E2 28211.075} C_VEL
LIN {X 0,Y 591.968,Z 353.055,A -85,B 0,C 180,E1 28207.693,E2 28207.693} C_VEL
LIN {X 0,Y 591.981,Z 353.054,A -85,B 0,C 180,E1 28204.812,E2 28204.812} C_VEL
LIN {X 0,Y 591.965,Z 353.055,A -85,B 0,C 180,E1 28201.575,E2 28201.575} C_VEL
LIN {X 0,Y 591.991,Z 353.054,A -85,B 0,C 180,E1 28198.664,E2 28198.664} C_VEL
LIN {X 0,Y 591.964,Z 353.055,A -85,B 0,C 180,E1 28195.513,E2 28195.513} C_VEL
LIN {X 0,Y 591.985,Z 353.054,A -85,B 0,C 180,E1 28192.65,E2 28192.65} C_VEL
LIN {X 0,Y 591.963,Z 353.055,A -85,B 0,C 180,E1 28189.436,E2 28189.436} C_VEL
LIN {X 0,Y 591.996,Z 353.053,A -85,B 0,C 180,E1 28186.484,E2 28186.484} C_VEL
LIN {X 0,Y 591.963,Z 353.054,A -85,B 0,C 180,E1 28183.369,E2 28183.369} C_VEL
LIN {X 0,Y 591.986,Z 353.054,A -85,B 0,C 180,E1 28180.51,E2 28180.51} C_VEL
LIN {X 0,Y 591.961,Z 353.055,A -85,B 0,C 180,E1 28177.278,E2 28177.278} C_VEL
LIN {X 0,Y 591.995,Z 353.054,A -85,B 0,C 180,E1 28174.359,E2 28174.359} C_VEL
LIN {X 0,Y 591.957,Z 353.055,A -85,B 0,C 180,E1 28171.161,E2 28171.161} C_VEL
LIN {X 0,Y 591.999,Z 353.053,A -85,B 0,C 180,E1 28168.258,E2 28168.258} C_VEL
LIN {X 0,Y 591.96,Z 353.055,A -85,B 0,C 180,E1 28165.155,E2 28165.155} C_VEL
LIN {X 0,Y 591.994,Z 353.053,A -85,B 0,C 180,E1 28162.235,E2 28162.235} C_VEL
LIN {X 0,Y 591.96,Z 353.055,A -85,B 0,C 180,E1 28159.095,E2 28159.095} C_VEL
LIN {X 0,Y 591.998,Z 353.054,A -85,B 0,C 180,E1 28156.123,E2 28156.123} C_VEL
LIN {X 0,Y 591.957,Z 353.055,A -85,B 0,C 180,E1 28152.944,E2 28152.944} C_VEL
LIN {X 0,Y 592.01,Z 353.055,A -85,B 0,C 180,E1 28149.949,E2 28149.949} C_VEL
LIN {X 0,Y 591.959,Z 353.055,A -85,B 0,C 180,E1 28146.929,E2 28146.929} C_VEL
LIN {X 0,Y 592.003,Z 353.054,A -85,B 0,C 180,E1 28143.952,E2 28143.952} C_VEL
LIN {X 0,Y 591.955,Z 353.055,A -85,B 0,C 180,E1 28140.781,E2 28140.781} C_VEL
LIN {X 0,Y 592.014,Z 353.055,A -85,B 0,C 180,E1 28137.795,E2 28137.795} C_VEL
LIN {X 0,Y 591.954,Z 353.055,A -85,B 0,C 180,E1 28134.67,E2 28134.67} C_VEL
LIN {X 0,Y 592.037,Z 353.055,A -85,B 0,C 180,E1 28131.574,E2 28131.574} C_VEL
LIN {X 0,Y 591.953,Z 353.055,A -85,B 0,C 180,E1 28128.538,E2 28128.538} C_VEL
LIN {X 0,Y 592.035,Z 353.056,A -85,B 0,C 180,E1 28125.455,E2 28125.455} C_VEL
LIN {X 0,Y 591.954,Z 353.055,A -85,B 0,C 180,E1 28122.372,E2 28122.372} C_VEL
LIN {X 0,Y 592.024,Z 353.056,A -85,B 0,C 180,E1 28119.297,E2 28119.297} C_VEL
LIN {X 0,Y 591.953,Z 353.055,A -85,B 0,C 180,E1 28116.322,E2 28116.322} C_VEL
LIN {X 0,Y 592.026,Z 353.057,A -85,B 0,C 180,E1 28113.28,E2 28113.28} C_VEL
LIN {X 0,Y 591.953,Z 353.056,A -85,B 0,C 180,E1 28110.222,E2 28110.222} C_VEL
LIN {X 0,Y 592.016,Z 353.05,A -85,B 0,C 180,E1 28107.119,E2 28107.119} C_VEL
LIN {X 0,Y 592.001,Z 353.174,A -85,B 0,C 180,E1 28106.886,E2 28106.886} C_VEL
LIN {X 0,Y 592.616,Z 357.515,A -85,B 0,C 180,E1 28106.375,E2 28106.375} C_VEL
LIN {X 0,Y 592.5,Z 386.083,A -85,B 0,C 180,E1 28103.259,E2 28103.259} C_VEL
LIN {X 0,Y 592.372,Z 415.335,A -85,B 0,C 180,E1 28100.141,E2 28100.141} C_VEL
LIN {X 0,Y 592.24,Z 447.195,A -85,B 0,C 180,E1 28096.813,E2 28096.813} C_VEL
LIN {X 0,Y 592.113,Z 478.719,A -85,B 0,C 180,E1 28093.575,E2 28093.575} C_VEL
LIN {X 0,Y 592.165,Z 481.138,A -85,B 0,C 180,E1 28093.361,E2 28093.361} C_VEL
LIN {X 0,Y 592.199,Z 592.411,A -85,B 0,C 180,E1 28091.979,E2 28091.979} C_VEL
LIN {X 0,Y 592.188,Z 607.141,A -85,B 0,C 180,E1 28091.618,E2 28091.618} C_VEL
LIN {X 0,Y 592.159,Z 620.9,A -85,B 0,C 180,E1 28091.098,E2 28091.098} C_VEL
LIN {X 0,Y 592.075,Z 634.339,A -85,B 0,C 180,E1 28090.41,E2 28090.41} C_VEL
LIN {X 0,Y 592.053,Z 647.296,A -85,B 0,C 180,E1 28089.527,E2 28089.527} C_VEL
LIN {X 0,Y 592.009,Z 658.505,A -85,B 0,C 180,E1 28088.547,E2 28088.547} C_VEL
LIN {X 0,Y 591.969,Z 668.219,A -85,B 0,C 180,E1 28087.473,E2 28087.473} C_VEL
LIN {X 0,Y 591.944,Z 676.55,A -85,B 0,C 180,E1 28086.303,E2 28086.303} C_VEL
LIN {X 0,Y 591.929,Z 683.488,A -85,B 0,C 180,E1 28085.039,E2 28085.039} C_VEL
LIN {X 0,Y 591.919,Z 688.938,A -85,B 0,C 180,E1 28083.68,E2 28083.68} C_VEL
LIN {X 0,Y 591.916,Z 692.766,A -85,B 0,C 180,E1 28082.227,E2 28082.227} C_VEL
LIN {X 0,Y 591.918,Z 694.69,A -85,B 0,C 180,E1 28080.774,E2 28080.774} C_VEL
LIN {X 0,Y 591.914,Z 694.813,A -85,B 0,C 180,E1 28079.323,E2 28079.323} C_VEL
LIN {X 0,Y 591.917,Z 692.956,A -85,B 0,C 180,E1 28077.774,E2 28077.774} C_VEL
LIN {X 0,Y 591.921,Z 689.224,A -85,B 0,C 180,E1 28076.32,E2 28076.32} C_VEL
LIN {X 0,Y 591.927,Z 683.915,A -85,B 0,C 180,E1 28074.961,E2 28074.961} C_VEL
LIN {X 0,Y 591.943,Z 677.123,A -85,B 0,C 180,E1 28073.697,E2 28073.697} C_VEL
LIN {X 0,Y 591.967,Z 668.83,A -85,B 0,C 180,E1 28072.514,E2 28072.514} C_VEL
LIN {X 0,Y 592.008,Z 658.426,A -85,B 0,C 180,E1 28071.355,E2 28071.355} C_VEL
LIN {X 0,Y 592.056,Z 647.196,A -85,B 0,C 180,E1 28070.376,E2 28070.376} C_VEL
LIN {X 0,Y 592.085,Z 634.206,A -85,B 0,C 180,E1 28069.492,E2 28069.492} C_VEL
LIN {X 0,Y 592.161,Z 620.71,A -85,B 0,C 180,E1 28068.803,E2 28068.803} C_VEL
LIN {X 0,Y 592.209,Z 606.954,A -85,B 0,C 180,E1 28068.286,E2 28068.286} C_VEL
LIN {X 0,Y 592.242,Z 591.174,A -85,B 0,C 180,E1 28067.91,E2 28067.91} C_VEL
LIN {X 0,Y 592.123,Z 480.688,A -85,B 0,C 180,E1 28066.536,E2 28066.536} C_VEL
LIN {X 0,Y 592.223,Z 448.873,A -85,B 0,C 180,E1 28063.27,E2 28063.27} C_VEL
LIN {X 0,Y 592.369,Z 417.653,A -85,B 0,C 180,E1 28060.014,E2 28060.014} C_VEL
LIN {X 0,Y 592.478,Z 388.29,A -85,B 0,C 180,E1 28056.888,E2 28056.888} C_VEL
LIN {X 0,Y 592.618,Z 358.645,A -85,B 0,C 180,E1 28053.658,E2 28053.658} C_VEL
LIN {X 0,Y 592.251,Z 354.355,A -85,B 0,C 180,E1 28053.153,E2 28053.153} C_VEL
LIN {X 0,Y 591.998,Z 353.06,A -85,B 0,C 180,E1 28052.978,E2 28052.978} C_VEL
LIN {X 0,Y 591.958,Z 353.057,A -85,B 0,C 180,E1 28049.861,E2 28049.861} C_VEL
LIN {X 0,Y 591.993,Z 353.056,A -85,B 0,C 180,E1 28046.939,E2 28046.939} C_VEL
LIN {X 0,Y 591.958,Z 353.056,A -85,B 0,C 180,E1 28043.76,E2 28043.76} C_VEL
LIN {X 0,Y 592.001,Z 353.055,A -85,B 0,C 180,E1 28040.826,E2 28040.826} C_VEL
LIN {X 0,Y 591.96,Z 353.055,A -85,B 0,C 180,E1 28037.716,E2 28037.716} C_VEL
LIN {X 0,Y 591.998,Z 353.055,A -85,B 0,C 180,E1 28034.773,E2 28034.773} C_VEL
LIN {X 0,Y 591.958,Z 353.056,A -85,B 0,C 180,E1 28031.591,E2 28031.591} C_VEL
LIN {X 0,Y 592.003,Z 353.055,A -85,B 0,C 180,E1 28028.676,E2 28028.676} C_VEL
LIN {X 0,Y 591.958,Z 353.056,A -85,B 0,C 180,E1 28025.498,E2 28025.498} C_VEL
LIN {X 0,Y 592.021,Z 353.056,A -85,B 0,C 180,E1 28022.484,E2 28022.484} C_VEL
LIN {X 0,Y 592.051,Z 353.298,A -85,B 0,C 180,E1 28020.487,E2 28020.487} C_VEL
LIN {X 0,Y 593.321,Z 357.886,A -85,B 0,C 180,E1 28020.089,E2 28020.089} C_VEL
LIN {X 0,Y 593.124,Z 398.843,A -85,B 0,C 180,E1 28017.238,E2 28017.238} C_VEL
LIN {X 0,Y 592.86,Z 445.314,A -85,B 0,C 180,E1 28014.088,E2 28014.088} C_VEL
LIN {X 0,Y 592.853,Z 463.125,A -85,B 0,C 180,E1 28012.923,E2 28012.923} C_VEL
LIN {X 0,Y 593.115,Z 474.869,A -85,B 0,C 180,E1 28012.761,E2 28012.761} C_VEL
LIN {X 0,Y 592.85,Z 672.313,A -85,B 0,C 180,E1 28010.227,E2 28010.227} C_VEL
LIN {X 0,Y 592.775,Z 691.305,A -85,B 0,C 180,E1 28009.797,E2 28009.797} C_VEL
LIN {X 0,Y 592.677,Z 709.402,A -85,B 0,C 180,E1 28009.206,E2 28009.206} C_VEL
LIN {X 0,Y 592.567,Z 727.05,A -85,B 0,C 180,E1 28008.444,E2 28008.444} C_VEL
LIN {X 0,Y 592.459,Z 743.694,A -85,B 0,C 180,E1 28007.538,E2 28007.538} C_VEL
LIN {X 0,Y 592.342,Z 759.637,A -85,B 0,C 180,E1 28006.474,E2 28006.474} C_VEL
LIN {X 0,Y 592.23,Z 774.562,A -85,B 0,C 180,E1 28005.27,E2 28005.27} C_VEL
LIN {X 0,Y 592.131,Z 788.018,A -85,B 0,C 180,E1 28003.973,E2 28003.973} C_VEL
LIN {X 0,Y 592.057,Z 800.418,A -85,B 0,C 180,E1 28002.547,E2 28002.547} C_VEL
LIN {X 0,Y 592.002,Z 811.588,A -85,B 0,C 180,E1 28001.003,E2 28001.003} C_VEL
LIN {X 0,Y 591.96,Z 821.474,A -85,B 0,C 180,E1 27999.332,E2 27999.332} C_VEL
LIN {X 0,Y 591.937,Z 829.773,A -85,B 0,C 180,E1 27997.571,E2 27997.571} C_VEL
LIN {X 0,Y 591.914,Z 836.259,A -85,B 0,C 180,E1 27995.769,E2 27995.769} C_VEL
LIN {X 0,Y 591.917,Z 840.874,A -85,B 0,C 180,E1 27993.971,E2 27993.971} C_VEL
LIN {X 0,Y 591.911,Z 843.788,A -85,B 0,C 180,E1 27992.13,E2 27992.13} C_VEL
LIN {X 0,Y 591.907,Z 844.94,A -85,B 0,C 180,E1 27990.29,E2 27990.29} C_VEL
LIN {X 0,Y 591.914,Z 844.349,A -85,B 0,C 180,E1 27988.451,E2 27988.451} C_VEL
LIN {X 0,Y 591.907,Z 842.006,A -85,B 0,C 180,E1 27986.611,E2 27986.611} C_VEL
LIN {X 0,Y 591.921,Z 838.097,A -85,B 0,C 180,E1 27984.864,E2 27984.864} C_VEL
LIN {X 0,Y 591.93,Z 832.466,A -85,B 0,C 180,E1 27983.112,E2 27983.112} C_VEL
LIN {X 0,Y 591.94,Z 825.424,A -85,B 0,C 180,E1 27981.452,E2 27981.452} C_VEL
LIN {X 0,Y 591.977,Z 816.511,A -85,B 0,C 180,E1 27979.785,E2 27979.785} C_VEL
LIN {X 0,Y 592.024,Z 806.146,A -85,B 0,C 180,E1 27978.208,E2 27978.208} C_VEL
LIN {X 0,Y 592.095,Z 794.346,A -85,B 0,C 180,E1 27976.723,E2 27976.723} C_VEL
LIN {X 0,Y 592.192,Z 780.579,A -85,B 0,C 180,E1 27975.279,E2 27975.279} C_VEL
LIN {X 0,Y 592.305,Z 765.593,A -85,B 0,C 180,E1 27973.978,E2 27973.978} C_VEL
LIN {X 0,Y 592.421,Z 749.418,A -85,B 0,C 180,E1 27972.821,E2 27972.821} C_VEL
LIN {X 0,Y 592.533,Z 733.034,A -85,B 0,C 180,E1 27971.86,E2 27971.86} C_VEL
LIN {X 0,Y 592.648,Z 716.134,A -85,B 0,C 180,E1 27971.062,E2 27971.062} C_VEL
LIN {X 0,Y 592.751,Z 697.83,A -85,B 0,C 180,E1 27970.396,E2 27970.396} C_VEL
LIN {X 0,Y 592.829,Z 679.294,A -85,B 0,C 180,E1 27969.911,E2 27969.911} C_VEL
LIN {X 0,Y 592.88,Z 659.503,A -85,B 0,C 180,E1 27969.586,E2 27969.586} C_VEL
LIN {X 0,Y 592.975,Z 463.898,A -85,B 0,C 180,E1 27967.092,E2 27967.092} C_VEL
LIN {X 0,Y 592.785,Z 461.934,A -85,B 0,C 180,E1 27967.021,E2 27967.021} C_VEL
LIN {X 0,Y 593.015,Z 416.251,A -85,B 0,C 180,E1 27963.951,E2 27963.951} C_VEL
LIN {X 0,Y 593.267,Z 372.851,A -85,B 0,C 180,E1 27960.963,E2 27960.963} C_VEL
LIN {X 0,Y 593.226,Z 356.985,A -85,B 0,C 180,E1 27959.842,E2 27959.842} C_VEL
LIN {X 0,Y 592.009,Z 353.043,A -85,B 0,C 180,E1 27959.469,E2 27959.469} C_VEL
LIN {X 0,Y 591.96,Z 353.056,A -85,B 0,C 180,E1 27956.473,E2 27956.473} C_VEL
LIN {X 0,Y 591.994,Z 353.054,A -85,B 0,C 180,E1 27953.28,E2 27953.28} C_VEL
LIN {X 0,Y 591.961,Z 353.055,A -85,B 0,C 180,E1 27950.373,E2 27950.373} C_VEL
LIN {X 0,Y 591.986,Z 353.055,A -85,B 0,C 180,E1 27947.14,E2 27947.14} C_VEL
LIN {X 0,Y 591.96,Z 353.055,A -85,B 0,C 180,E1 27944.261,E2 27944.261} C_VEL
LIN {X 0,Y 591.976,Z 353.055,A -85,B 0,C 180,E1 27940.975,E2 27940.975} C_VEL
LIN {X 0,Y 591.96,Z 353.056,A -85,B 0,C 180,E1 27938.185,E2 27938.185} C_VEL
LIN {X 0,Y 591.977,Z 353.056,A -85,B 0,C 180,E1 27934.93,E2 27934.93} C_VEL
LIN {X 0,Y 591.959,Z 353.056,A -85,B 0,C 180,E1 27932.144,E2 27932.144} C_VEL
LIN {X 0,Y 591.98,Z 353.057,A -85,B 0,C 180,E1 27928.885,E2 27928.885} C_VEL
LIN {X 0,Y 592.041,Z 353.204,A -85,B 0,C 180,E1 27927.223,E2 27927.223} C_VEL
LIN {X 0,Y 592.851,Z 357.041,A -85,B 0,C 180,E1 27926.852,E2 27926.852} C_VEL
LIN {X 0,Y 592.725,Z 391.989,A -85,B 0,C 180,E1 27923.882,E2 27923.882} C_VEL
LIN {X 0,Y 592.723,Z 404.426,A -85,B 0,C 180,E1 27922.866,E2 27922.866} C_VEL
LIN {X 0,Y 593.093,Z 409.609,A -85,B 0,C 180,E1 27922.785,E2 27922.785} C_VEL
LIN {X 0,Y 592.849,Z 612.53,A -85,B 0,C 180,E1 27920.179,E2 27920.179} C_VEL
LIN {X 0,Y 592.771,Z 631.882,A -85,B 0,C 180,E1 27919.737,E2 27919.737} C_VEL
LIN {X 0,Y 592.669,Z 650.096,A -85,B 0,C 180,E1 27919.135,E2 27919.135} C_VEL
LIN {X 0,Y 592.56,Z 667.892,A -85,B 0,C 180,E1 27918.358,E2 27918.358} C_VEL
LIN {X 0,Y 592.446,Z 684.703,A -85,B 0,C 180,E1 27917.431,E2 27917.431} C_VEL
LIN {X 0,Y 592.327,Z 700.74,A -85,B 0,C 180,E1 27916.347,E2 27916.347} C_VEL
LIN {X 0,Y 592.215,Z 715.714,A -85,B 0,C 180,E1 27915.12,E2 27915.12} C_VEL
LIN {X 0,Y 592.13,Z 729.469,A -85,B 0,C 180,E1 27913.774,E2 27913.774} C_VEL
LIN {X 0,Y 592.052,Z 742.113,A -85,B 0,C 180,E1 27912.286,E2 27912.286} C_VEL
LIN {X 0,Y 591.992,Z 753.21,A -85,B 0,C 180,E1 27910.707,E2 27910.707} C_VEL
LIN {X 0,Y 591.958,Z 762.797,A -85,B 0,C 180,E1 27909.038,E2 27909.038} C_VEL
LIN {X 0,Y 591.935,Z 770.405,A -85,B 0,C 180,E1 27907.376,E2 27907.376} C_VEL
LIN {X 0,Y 591.923,Z 776.571,A -85,B 0,C 180,E1 27905.622,E2 27905.622} C_VEL
LIN {X 0,Y 591.918,Z 781.192,A -85,B 0,C 180,E1 27903.777,E2 27903.777} C_VEL
LIN {X 0,Y 591.908,Z 783.966,A -85,B 0,C 180,E1 27901.936,E2 27901.936} C_VEL
LIN {X 0,Y 591.911,Z 784.974,A -85,B 0,C 180,E1 27900.097,E2 27900.097} C_VEL
LIN {X 0,Y 591.908,Z 784.242,A -85,B 0,C 180,E1 27898.257,E2 27898.257} C_VEL
LIN {X 0,Y 591.908,Z 781.762,A -85,B 0,C 180,E1 27896.416,E2 27896.416} C_VEL
LIN {X 0,Y 591.919,Z 777.448,A -85,B 0,C 180,E1 27894.572,E2 27894.572} C_VEL
LIN {X 0,Y 591.928,Z 771.182,A -85,B 0,C 180,E1 27892.722,E2 27892.722} C_VEL
LIN {X 0,Y 591.958,Z 763.268,A -85,B 0,C 180,E1 27890.962,E2 27890.962} C_VEL
LIN {X 0,Y 591.959,Z 760.581,A -85,B 0,C 180,E1 27890.452,E2 27890.452} C_VEL
LIN {X 0,Y 591.009,Z 757.029,A -85,B 0,C 180,E1 27889.79,E2 27889.79} C_VEL
LIN {X 0,Y 585.963,Z 749.07,A -85,B 0,C 180,E1 27888.435,E2 27888.435} C_VEL
LIN {X 0,Y 584.21,Z 744.176,A -85,B 0,C 180,E1 27887.725,E2 27887.725} C_VEL
LIN {X 0,Y 584.121,Z 742.851,A -85,B 0,C 180,E1 27887.549,E2 27887.549} C_VEL
LIN {X 0,Y 584.235,Z 730.13,A -85,B 0,C 180,E1 27886.017,E2 27886.017} C_VEL
LIN {X 0,Y 584.375,Z 716.145,A -85,B 0,C 180,E1 27884.621,E2 27884.621} C_VEL
LIN {X 0,Y 584.55,Z 700.837,A -85,B 0,C 180,E1 27883.346,E2 27883.346} C_VEL
LIN {X 0,Y 584.735,Z 684.506,A -85,B 0,C 180,E1 27882.228,E2 27882.228} C_VEL
LIN {X 0,Y 584.918,Z 667.159,A -85,B 0,C 180,E1 27881.265,E2 27881.265} C_VEL
LIN {X 0,Y 585.1,Z 648.589,A -85,B 0,C 180,E1 27880.457,E2 27880.457} C_VEL
LIN {X 0,Y 585.244,Z 629.363,A -85,B 0,C 180,E1 27879.838,E2 27879.838} C_VEL
LIN {X 0,Y 585.349,Z 610.405,A -85,B 0,C 180,E1 27879.425,E2 27879.425} C_VEL
LIN {X 0,Y 585.584,Z 406.897,A -85,B 0,C 180,E1 27876.78,E2 27876.78} C_VEL
LIN {X 0,Y 585.061,Z 403.734,A -85,B 0,C 180,E1 27876.695,E2 27876.695} C_VEL
LIN {X 0,Y 585.327,Z 367.276,A -85,B 0,C 180,E1 27873.577,E2 27873.577} C_VEL
LIN {X 0,Y 585.309,Z 358.477,A -85,B 0,C 180,E1 27872.809,E2 27872.809} C_VEL
LIN {X 0,Y 584.065,Z 354.047,A -85,B 0,C 180,E1 27872.332,E2 27872.332} C_VEL
LIN {X 0,Y 584.027,Z 354.045,A -85,B 0,C 180,E1 27869.324,E2 27869.324} C_VEL
LIN {X 0,Y 584.044,Z 354.045,A -85,B 0,C 180,E1 27866.075,E2 27866.075} C_VEL
LIN {X 0,Y 584.03,Z 354.044,A -85,B 0,C 180,E1 27863.187,E2 27863.187} C_VEL
LIN {X 0,Y 584.028,Z 354.044,A -85,B 0,C 180,E1 27859.802,E2 27859.802} C_VEL
LIN {X 0,Y 584.057,Z 354.043,A -85,B 0,C 180,E1 27856.826,E2 27856.826} C_VEL
LIN {X 0,Y 584.023,Z 354.044,A -85,B 0,C 180,E1 27853.599,E2 27853.599} C_VEL
LIN {X 0,Y 584.094,Z 354.043,A -85,B 0,C 180,E1 27850.45,E2 27850.45} C_VEL
LIN {X 0,Y 584.02,Z 354.044,A -85,B 0,C 180,E1 27847.403,E2 27847.403} C_VEL
LIN {X 0,Y 584.094,Z 354.045,A -85,B 0,C 180,E1 27844.277,E2 27844.277} C_VEL
LIN {X 0,Y 584.021,Z 354.043,A -85,B 0,C 180,E1 27841.128,E2 27841.128} C_VEL
LIN {X 0,Y 584.062,Z 354.044,A -85,B 0,C 180,E1 27837.951,E2 27837.951} C_VEL
LIN {X 0,Y 584.023,Z 354.043,A -85,B 0,C 180,E1 27835.016,E2 27835.016} C_VEL
LIN {X 0,Y 584.052,Z 354.044,A -85,B 0,C 180,E1 27831.808,E2 27831.808} C_VEL
LIN {X 0,Y 584.025,Z 354.043,A -85,B 0,C 180,E1 27828.879,E2 27828.879} C_VEL
LIN {X 0,Y 584.037,Z 354.044,A -85,B 0,C 180,E1 27825.592,E2 27825.592} C_VEL
LIN {X 0,Y 584.028,Z 354.043,A -85,B 0,C 180,E1 27822.759,E2 27822.759} C_VEL
LIN {X 0,Y 584.032,Z 354.043,A -85,B 0,C 180,E1 27819.46,E2 27819.46} C_VEL
LIN {X 0,Y 584.035,Z 354.043,A -85,B 0,C 180,E1 27816.587,E2 27816.587} C_VEL
LIN {X 0,Y 584.027,Z 354.043,A -85,B 0,C 180,E1 27813.337,E2 27813.337} C_VEL
LIN {X 0,Y 584.037,Z 354.043,A -85,B 0,C 180,E1 27810.49,E2 27810.49} C_VEL
LIN {X 0,Y 584.026,Z 354.043,A -85,B 0,C 180,E1 27807.252,E2 27807.252} C_VEL
LIN {X 0,Y 584.048,Z 354.043,A -85,B 0,C 180,E1 27804.302,E2 27804.302} C_VEL
LIN {X 0,Y 584.02,Z 354.043,A -85,B 0,C 180,E1 27801.057,E2 27801.057} C_VEL
LIN {X 0,Y 584.072,Z 354.043,A -85,B 0,C 180,E1 27798.045,E2 27798.045} C_VEL
LIN {X 0,Y 584.018,Z 354.044,A -85,B 0,C 180,E1 27794.916,E2 27794.916} C_VEL
LIN {X 0,Y 584.092,Z 354.043,A -85,B 0,C 180,E1 27791.817,E2 27791.817} C_VEL
LIN {X 0,Y 584.016,Z 354.044,A -85,B 0,C 180,E1 27788.718,E2 27788.718} C_VEL
LIN {X 0,Y 584.085,Z 354.045,A -85,B 0,C 180,E1 27785.603,E2 27785.603} C_VEL
LIN {X 0,Y 584.016,Z 354.044,A -85,B 0,C 180,E1 27782.578,E2 27782.578} C_VEL
LIN {X 0,Y 584.075,Z 354.044,A -85,B 0,C 180,E1 27779.437,E2 27779.437} C_VEL
LIN {X 0,Y 584.017,Z 354.044,A -85,B 0,C 180,E1 27776.427,E2 27776.427} C_VEL
LIN {X 0,Y 584.051,Z 354.045,A -85,B 0,C 180,E1 27773.189,E2 27773.189} C_VEL
LIN {X 0,Y 584.019,Z 354.044,A -85,B 0,C 180,E1 27770.313,E2 27770.313} C_VEL
LIN {X 0,Y 584.043,Z 354.044,A -85,B 0,C 180,E1 27767.05,E2 27767.05} C_VEL
LIN {X 0,Y 584.022,Z 354.044,A -85,B 0,C 180,E1 27764.165,E2 27764.165} C_VEL
LIN {X 0,Y 584.028,Z 354.045,A -85,B 0,C 180,E1 27760.825,E2 27760.825} C_VEL
LIN {X 0,Y 584.025,Z 354.044,A -85,B 0,C 180,E1 27758.045,E2 27758.045} C_VEL
LIN {X 0,Y 584.026,Z 354.045,A -85,B 0,C 180,E1 27754.738,E2 27754.738} C_VEL
LIN {X 0,Y 584.037,Z 354.045,A -85,B 0,C 180,E1 27751.823,E2 27751.823} C_VEL
LIN {X 0,Y 584.018,Z 354.047,A -85,B 0,C 180,E1 27748.533,E2 27748.533} C_VEL
LIN {X 0,Y 584.1,Z 354.174,A -85,B 0,C 180,E1 27747.167,E2 27747.167} C_VEL
LIN {X 0,Y 585.016,Z 359.283,A -85,B 0,C 180,E1 27746.547,E2 27746.547} C_VEL
LIN {X 0,Y 584.815,Z 387.552,A -85,B 0,C 180,E1 27743.422,E2 27743.422} C_VEL
LIN {X 0,Y 584.61,Z 416.874,A -85,B 0,C 180,E1 27740.256,E2 27740.256} C_VEL
LIN {X 0,Y 584.405,Z 448.495,A -85,B 0,C 180,E1 27736.909,E2 27736.909} C_VEL
LIN {X 0,Y 584.223,Z 479.7,A -85,B 0,C 180,E1 27733.661,E2 27733.661} C_VEL
LIN {X 0,Y 584.28,Z 481.232,A -85,B 0,C 180,E1 27733.544,E2 27733.544} C_VEL
LIN {X 0,Y 584.532,Z 500.368,A -85,B 0,C 180,E1 27733.301,E2 27733.301} C_VEL
LIN {X 0,Y 584.371,Z 592.46,A -85,B 0,C 180,E1 27732.142,E2 27732.142} C_VEL
LIN {X 0,Y 584.335,Z 607.96,A -85,B 0,C 180,E1 27731.749,E2 27731.749} C_VEL
LIN {X 0,Y 584.283,Z 622.014,A -85,B 0,C 180,E1 27731.2,E2 27731.2} C_VEL
LIN {X 0,Y 584.17,Z 635.157,A -85,B 0,C 180,E1 27730.503,E2 27730.503} C_VEL
LIN {X 0,Y 584.122,Z 647.289,A -85,B 0,C 180,E1 27729.657,E2 27729.657} C_VEL
LIN {X 0,Y 584.055,Z 658.51,A -85,B 0,C 180,E1 27728.665,E2 27728.665} C_VEL
LIN {X 0,Y 583.994,Z 668.998,A -85,B 0,C 180,E1 27727.477,E2 27727.477} C_VEL
LIN {X 0,Y 583.957,Z 677.161,A -85,B 0,C 180,E1 27726.291,E2 27726.291} C_VEL
LIN {X 0,Y 583.934,Z 684.408,A -85,B 0,C 180,E1 27724.911,E2 27724.911} C_VEL
LIN {X 0,Y 583.92,Z 689.546,A -85,B 0,C 180,E1 27723.534,E2 27723.534} C_VEL
LIN {X 0,Y 583.917,Z 692.969,A -85,B 0,C 180,E1 27722.159,E2 27722.159} C_VEL
LIN {X 0,Y 583.918,Z 694.757,A -85,B 0,C 180,E1 27720.687,E2 27720.687} C_VEL
LIN {X 0,Y 583.914,Z 694.752,A -85,B 0,C 180,E1 27719.215,E2 27719.215} C_VEL
LIN {X 0,Y 583.917,Z 692.952,A -85,B 0,C 180,E1 27717.743,E2 27717.743} C_VEL
LIN {X 0,Y 583.922,Z 689.214,A -85,B 0,C 180,E1 27716.269,E2 27716.269} C_VEL
LIN {X 0,Y 583.934,Z 683.915,A -85,B 0,C 180,E1 27714.892,E2 27714.892} C_VEL
LIN {X 0,Y 583.957,Z 677.108,A -85,B 0,C 180,E1 27713.61,E2 27713.61} C_VEL
LIN {X 0,Y 583.994,Z 668.93,A -85,B 0,C 180,E1 27712.425,E2 27712.425} C_VEL
LIN {X 0,Y 584.056,Z 658.419,A -85,B 0,C 180,E1 27711.236,E2 27711.236} C_VEL
LIN {X 0,Y 584.127,Z 647.173,A -85,B 0,C 180,E1 27710.244,E2 27710.244} C_VEL
LIN {X 0,Y 584.19,Z 634.199,A -85,B 0,C 180,E1 27709.348,E2 27709.348} C_VEL
LIN {X 0,Y 584.287,Z 621.362,A -85,B 0,C 180,E1 27708.681,E2 27708.681} C_VEL
LIN {X 0,Y 584.356,Z 607.669,A -85,B 0,C 180,E1 27708.152,E2 27708.152} C_VEL
LIN {X 0,Y 584.415,Z 592.013,A -85,B 0,C 180,E1 27707.761,E2 27707.761} C_VEL
LIN {X 0,Y 584.315,Z 481.458,A -85,B 0,C 180,E1 27706.37,E2 27706.37} C_VEL
LIN {X 0,Y 584.233,Z 480.572,A -85,B 0,C 180,E1 27706.339,E2 27706.339} C_VEL
LIN {X 0,Y 584.39,Z 449.354,A -85,B 0,C 180,E1 27703.091,E2 27703.091} C_VEL
LIN {X 0,Y 584.602,Z 418.989,A -85,B 0,C 180,E1 27699.88,E2 27699.88} C_VEL
LIN {X 0,Y 584.786,Z 389.84,A -85,B 0,C 180,E1 27696.737,E2 27696.737} C_VEL
LIN {X 0,Y 585.078,Z 360.874,A -85,B 0,C 180,E1 27693.511,E2 27693.511} C_VEL
LIN {X 0,Y 584.781,Z 357.06,A -85,B 0,C 180,E1 27693.058,E2 27693.058} C_VEL
LIN {X 0,Y 584.088,Z 354.046,A -85,B 0,C 180,E1 27692.637,E2 27692.637} C_VEL
LIN {X 0,Y 584.016,Z 354.046,A -85,B 0,C 180,E1 27689.552,E2 27689.552} C_VEL
LIN {X 0,Y 584.079,Z 354.046,A -85,B 0,C 180,E1 27686.432,E2 27686.432} C_VEL
LIN {X 0,Y 584.017,Z 354.045,A -85,B 0,C 180,E1 27683.413,E2 27683.413} C_VEL
LIN {X 0,Y 584.062,Z 354.045,A -85,B 0,C 180,E1 27680.233,E2 27680.233} C_VEL
LIN {X 0,Y 584.021,Z 354.044,A -85,B 0,C 180,E1 27677.262,E2 27677.262} C_VEL
LIN {X 0,Y 584.048,Z 354.045,A -85,B 0,C 180,E1 27674.027,E2 27674.027} C_VEL
LIN {X 0,Y 584.027,Z 354.044,A -85,B 0,C 180,E1 27671.103,E2 27671.103} C_VEL
LIN {X 0,Y 584.031,Z 354.045,A -85,B 0,C 180,E1 27667.726,E2 27667.726} C_VEL
LIN {X 0,Y 584.047,Z 354.045,A -85,B 0,C 180,E1 27664.756,E2 27664.756} C_VEL
LIN {X 0,Y 584.024,Z 354.048,A -85,B 0,C 180,E1 27661.506,E2 27661.506} C_VEL
LIN {X 0,Y 584.051,Z 354.176,A -85,B 0,C 180,E1 27660.886,E2 27660.886} C_VEL
LIN {X 0,Y 586.071,Z 360.453,A -85,B 0,C 180,E1 27660.316,E2 27660.316} C_VEL
LIN {X 0,Y 585.739,Z 401.915,A -85,B 0,C 180,E1 27657.395,E2 27657.395} C_VEL
LIN {X 0,Y 585.346,Z 447.798,A -85,B 0,C 180,E1 27654.248,E2 27654.248} C_VEL
LIN {X 0,Y 585.317,Z 463.159,A -85,B 0,C 180,E1 27653.235,E2 27653.235} C_VEL
LIN {X 0,Y 585.747,Z 469.016,A -85,B 0,C 180,E1 27653.14,E2 27653.14} C_VEL
LIN {X 0,Y 585.339,Z 672.313,A -85,B 0,C 180,E1 27650.498,E2 27650.498} C_VEL
LIN {X 0,Y 585.225,Z 691.348,A -85,B 0,C 180,E1 27650.062,E2 27650.062} C_VEL
LIN {X 0,Y 585.081,Z 709.399,A -85,B 0,C 180,E1 27649.466,E2 27649.466} C_VEL
LIN {X 0,Y 584.918,Z 726.946,A -85,B 0,C 180,E1 27648.699,E2 27648.699} C_VEL
LIN {X 0,Y 584.739,Z 744.215,A -85,B 0,C 180,E1 27647.744,E2 27647.744} C_VEL
LIN {X 0,Y 584.56,Z 760.235,A -85,B 0,C 180,E1 27646.654,E2 27646.654} C_VEL
LIN {X 0,Y 584.394,Z 775.089,A -85,B 0,C 180,E1 27645.432,E2 27645.432} C_VEL
LIN {X 0,Y 584.241,Z 788.944,A -85,B 0,C 180,E1 27644.065,E2 27644.065} C_VEL
LIN {X 0,Y 584.125,Z 801.684,A -85,B 0,C 180,E1 27642.556,E2 27642.556} C_VEL
LIN {X 0,Y 584.041,Z 812.866,A -85,B 0,C 180,E1 27640.955,E2 27640.955} C_VEL
LIN {X 0,Y 583.984,Z 822.509,A -85,B 0,C 180,E1 27639.262,E2 27639.262} C_VEL
LIN {X 0,Y 583.946,Z 830.391,A -85,B 0,C 180,E1 27637.524,E2 27637.524} C_VEL
LIN {X 0,Y 583.918,Z 836.411,A -85,B 0,C 180,E1 27635.798,E2 27635.798} C_VEL
LIN {X 0,Y 583.916,Z 840.874,A -85,B 0,C 180,E1 27634.026,E2 27634.026} C_VEL
LIN {X 0,Y 583.911,Z 843.789,A -85,B 0,C 180,E1 27632.159,E2 27632.159} C_VEL
LIN {X 0,Y 583.907,Z 844.94,A -85,B 0,C 180,E1 27630.294,E2 27630.294} C_VEL
LIN {X 0,Y 583.913,Z 844.349,A -85,B 0,C 180,E1 27628.43,E2 27628.43} C_VEL
LIN {X 0,Y 583.907,Z 842.006,A -85,B 0,C 180,E1 27626.564,E2 27626.564} C_VEL
LIN {X 0,Y 583.923,Z 838.097,A -85,B 0,C 180,E1 27624.793,E2 27624.793} C_VEL
LIN {X 0,Y 583.938,Z 832.466,A -85,B 0,C 180,E1 27623.017,E2 27623.017} C_VEL
LIN {X 0,Y 583.956,Z 825.424,A -85,B 0,C 180,E1 27621.334,E2 27621.334} C_VEL
LIN {X 0,Y 584.015,Z 816.512,A -85,B 0,C 180,E1 27619.644,E2 27619.644} C_VEL
LIN {X 0,Y 584.087,Z 806.147,A -85,B 0,C 180,E1 27618.046,E2 27618.046} C_VEL
LIN {X 0,Y 584.197,Z 794.347,A -85,B 0,C 180,E1 27616.54,E2 27616.54} C_VEL
LIN {X 0,Y 584.341,Z 780.578,A -85,B 0,C 180,E1 27615.077,E2 27615.077} C_VEL
LIN {X 0,Y 584.508,Z 765.596,A -85,B 0,C 180,E1 27613.759,E2 27613.759} C_VEL
LIN {X 0,Y 584.686,Z 749.42,A -85,B 0,C 180,E1 27612.587,E2 27612.587} C_VEL
LIN {X 0,Y 584.862,Z 732.526,A -85,B 0,C 180,E1 27611.588,E2 27611.588} C_VEL
LIN {X 0,Y 585.033,Z 715.797,A -85,B 0,C 180,E1 27610.792,E2 27610.792} C_VEL
LIN {X 0,Y 585.187,Z 697.727,A -85,B 0,C 180,E1 27610.129,E2 27610.129} C_VEL
LIN {X 0,Y 585.306,Z 679.131,A -85,B 0,C 180,E1 27609.638,E2 27609.638} C_VEL
LIN {X 0,Y 585.382,Z 659.277,A -85,B 0,C 180,E1 27609.31,E2 27609.31} C_VEL
LIN {X 0,Y 585.595,Z 464.915,A -85,B 0,C 180,E1 27606.8,E2 27606.8} C_VEL
LIN {X 0,Y 585.246,Z 462.249,A -85,B 0,C 180,E1 27606.729,E2 27606.729} C_VEL
LIN {X 0,Y 585.608,Z 416.172,A -85,B 0,C 180,E1 27603.591,E2 27603.591} C_VEL
LIN {X 0,Y 585.977,Z 373.639,A -85,B 0,C 180,E1 27600.622,E2 27600.622} C_VEL
LIN {X 0,Y 585.929,Z 359.553,A -85,B 0,C 180,E1 27599.611,E2 27599.611} C_VEL
LIN {X 0,Y 584.031,Z 354.032,A -85,B 0,C 180,E1 27599.096,E2 27599.096} C_VEL
LIN {X 0,Y 584.046,Z 354.046,A -85,B 0,C 180,E1 27596.129,E2 27596.129} C_VEL
LIN {X 0,Y 584.026,Z 354.044,A -85,B 0,C 180,E1 27592.92,E2 27592.92} C_VEL
LIN {X 0,Y 584.044,Z 354.045,A -85,B 0,C 180,E1 27590.06,E2 27590.06} C_VEL
LIN {X 0,Y 584.021,Z 354.044,A -85,B 0,C 180,E1 27586.779,E2 27586.779} C_VEL
LIN {X 0,Y 584.053,Z 354.045,A -85,B 0,C 180,E1 27583.885,E2 27583.885} C_VEL
LIN {X 0,Y 584.019,Z 354.044,A -85,B 0,C 180,E1 27580.674,E2 27580.674} C_VEL
LIN {X 0,Y 584.054,Z 354.045,A -85,B 0,C 180,E1 27577.797,E2 27577.797} C_VEL
LIN {X 0,Y 584.017,Z 354.045,A -85,B 0,C 180,E1 27574.564,E2 27574.564} C_VEL
LIN {X 0,Y 584.087,Z 354.047,A -85,B 0,C 180,E1 27571.474,E2 27571.474} C_VEL
LIN {X 0,Y 584.014,Z 354.047,A -85,B 0,C 180,E1 27568.358,E2 27568.358} C_VEL
LIN {X 0,Y 584.094,Z 354.23,A -85,B 0,C 180,E1 27567.536,E2 27567.536} C_VEL
LIN {X 0,Y 585.368,Z 359.335,A -85,B 0,C 180,E1 27567.023,E2 27567.023} C_VEL
LIN {X 0,Y 585.14,Z 393.882,A -85,B 0,C 180,E1 27564.05,E2 27564.05} C_VEL
LIN {X 0,Y 585.136,Z 404.513,A -85,B 0,C 180,E1 27563.18,E2 27563.18} C_VEL
LIN {X 0,Y 585.719,Z 409.604,A -85,B 0,C 180,E1 27563.089,E2 27563.089} C_VEL
LIN {X 0,Y 585.339,Z 612.402,A -85,B 0,C 180,E1 27560.452,E2 27560.452} C_VEL
LIN {X 0,Y 585.218,Z 631.836,A -85,B 0,C 180,E1 27560.004,E2 27560.004} C_VEL
LIN {X 0,Y 585.076,Z 649.724,A -85,B 0,C 180,E1 27559.409,E2 27559.409} C_VEL
LIN {X 0,Y 584.914,Z 667.212,A -85,B 0,C 180,E1 27558.642,E2 27558.642} C_VEL
LIN {X 0,Y 584.746,Z 683.894,A -85,B 0,C 180,E1 27557.72,E2 27557.72} C_VEL
LIN {X 0,Y 584.56,Z 700.406,A -85,B 0,C 180,E1 27556.597,E2 27556.597} C_VEL
LIN {X 0,Y 584.382,Z 715.718,A -85,B 0,C 180,E1 27555.328,E2 27555.328} C_VEL
LIN {X 0,Y 584.241,Z 729.48,A -85,B 0,C 180,E1 27553.963,E2 27553.963} C_VEL
LIN {X 0,Y 584.123,Z 742.121,A -85,B 0,C 180,E1 27552.455,E2 27552.455} C_VEL
LIN {X 0,Y 584.037,Z 753.213,A -85,B 0,C 180,E1 27550.855,E2 27550.855} C_VEL
LIN {X 0,Y 583.981,Z 762.804,A -85,B 0,C 180,E1 27549.162,E2 27549.162} C_VEL
LIN {X 0,Y 583.944,Z 770.817,A -85,B 0,C 180,E1 27547.378,E2 27547.378} C_VEL
LIN {X 0,Y 583.926,Z 776.875,A -85,B 0,C 180,E1 27545.601,E2 27545.601} C_VEL
LIN {X 0,Y 583.919,Z 781.392,A -85,B 0,C 180,E1 27543.731,E2 27543.731} C_VEL
LIN {X 0,Y 583.908,Z 784.079,A -85,B 0,C 180,E1 27541.864,E2 27541.864} C_VEL
LIN {X 0,Y 583.914,Z 784.996,A -85,B 0,C 180,E1 27540,E2 27540} C_VEL
LIN {X 0,Y 583.905,Z 784.156,A -85,B 0,C 180,E1 27538.135,E2 27538.135} C_VEL
LIN {X 0,Y 583.912,Z 781.566,A -85,B 0,C 180,E1 27536.269,E2 27536.269} C_VEL
LIN {X 0,Y 583.919,Z 777.15,A -85,B 0,C 180,E1 27534.399,E2 27534.399} C_VEL
LIN {X 0,Y 583.936,Z 771.18,A -85,B 0,C 180,E1 27532.622,E2 27532.622} C_VEL
LIN {X 0,Y 583.978,Z 763.259,A -85,B 0,C 180,E1 27530.838,E2 27530.838} C_VEL
LIN {X 0,Y 584.039,Z 753.782,A -85,B 0,C 180,E1 27529.145,E2 27529.145} C_VEL
LIN {X 0,Y 584.121,Z 742.851,A -85,B 0,C 180,E1 27527.549,E2 27527.549} C_VEL
LIN {X 0,Y 583.158,Z 738.309,A -85,B 0,C 180,E1 27526.944,E2 27526.944} C_VEL
LIN {X 0,Y 577.382,Z 726.431,A -85,B 0,C 180,E1 27525.444,E2 27525.444} C_VEL
LIN {X 0,Y 576.491,Z 721.126,A -85,B 0,C 180,E1 27524.879,E2 27524.879} C_VEL
LIN {X 0,Y 576.713,Z 706.085,A -85,B 0,C 180,E1 27523.528,E2 27523.528} C_VEL
LIN {X 0,Y 576.963,Z 689.335,A -85,B 0,C 180,E1 27522.294,E2 27522.294} C_VEL
LIN {X 0,Y 577.205,Z 671.933,A -85,B 0,C 180,E1 27521.256,E2 27521.256} C_VEL
LIN {X 0,Y 577.443,Z 654.368,A -85,B 0,C 180,E1 27520.424,E2 27520.424} C_VEL
LIN {X 0,Y 577.651,Z 635.328,A -85,B 0,C 180,E1 27519.737,E2 27519.737} C_VEL
LIN {X 0,Y 577.809,Z 616.201,A -85,B 0,C 180,E1 27519.256,E2 27519.256} C_VEL
LIN {X 0,Y 577.901,Z 592.251,A -85,B 0,C 180,E1 27518.892,E2 27518.892} C_VEL
LIN {X 0,Y 578.197,Z 407.878,A -85,B 0,C 180,E1 27516.48,E2 27516.48} C_VEL
LIN {X 0,Y 577.471,Z 403.725,A -85,B 0,C 180,E1 27516.37,E2 27516.37} C_VEL
LIN {X 0,Y 577.845,Z 366.639,A -85,B 0,C 180,E1 27513.152,E2 27513.152} C_VEL
LIN {X 0,Y 577.695,Z 360.598,A -85,B 0,C 180,E1 27512.61,E2 27512.61} C_VEL
LIN {X 0,Y 576.095,Z 355.037,A -85,B 0,C 180,E1 27512,E2 27512} C_VEL
LIN {X 0,Y 576.112,Z 355.034,A -85,B 0,C 180,E1 27509.021,E2 27509.021} C_VEL
LIN {X 0,Y 576.086,Z 355.034,A -85,B 0,C 180,E1 27505.782,E2 27505.782} C_VEL
LIN {X 0,Y 576.139,Z 355.032,A -85,B 0,C 180,E1 27502.723,E2 27502.723} C_VEL
LIN {X 0,Y 576.083,Z 355.033,A -85,B 0,C 180,E1 27499.636,E2 27499.636} C_VEL
LIN {X 0,Y 576.155,Z 355.033,A -85,B 0,C 180,E1 27496.502,E2 27496.502} C_VEL
LIN {X 0,Y 576.082,Z 355.032,A -85,B 0,C 180,E1 27493.345,E2 27493.345} C_VEL
LIN {X 0,Y 576.141,Z 355.033,A -85,B 0,C 180,E1 27490.21,E2 27490.21} C_VEL
LIN {X 0,Y 576.084,Z 355.032,A -85,B 0,C 180,E1 27487.157,E2 27487.157} C_VEL
LIN {X 0,Y 576.104,Z 355.033,A -85,B 0,C 180,E1 27483.857,E2 27483.857} C_VEL
LIN {X 0,Y 576.094,Z 355.032,A -85,B 0,C 180,E1 27480.913,E2 27480.913} C_VEL
LIN {X 0,Y 576.091,Z 355.033,A -85,B 0,C 180,E1 27477.607,E2 27477.607} C_VEL
LIN {X 0,Y 576.102,Z 355.032,A -85,B 0,C 180,E1 27474.726,E2 27474.726} C_VEL
LIN {X 0,Y 576.087,Z 355.032,A -85,B 0,C 180,E1 27471.482,E2 27471.482} C_VEL
LIN {X 0,Y 576.117,Z 355.032,A -85,B 0,C 180,E1 27468.518,E2 27468.518} C_VEL
LIN {X 0,Y 576.082,Z 355.033,A -85,B 0,C 180,E1 27465.297,E2 27465.297} C_VEL
LIN {X 0,Y 576.145,Z 355.031,A -85,B 0,C 180,E1 27462.223,E2 27462.223} C_VEL
LIN {X 0,Y 576.079,Z 355.032,A -85,B 0,C 180,E1 27459.041,E2 27459.041} C_VEL
LIN {X 0,Y 576.143,Z 355.033,A -85,B 0,C 180,E1 27455.877,E2 27455.877} C_VEL
LIN {X 0,Y 576.082,Z 355.032,A -85,B 0,C 180,E1 27452.786,E2 27452.786} C_VEL
LIN {X 0,Y 576.106,Z 355.032,A -85,B 0,C 180,E1 27449.503,E2 27449.503} C_VEL
LIN {X 0,Y 576.093,Z 355.031,A -85,B 0,C 180,E1 27446.517,E2 27446.517} C_VEL
LIN {X 0,Y 576.088,Z 355.032,A -85,B 0,C 180,E1 27443.222,E2 27443.222} C_VEL
LIN {X 0,Y 576.105,Z 355.032,A -85,B 0,C 180,E1 27440.308,E2 27440.308} C_VEL
LIN {X 0,Y 576.083,Z 355.032,A -85,B 0,C 180,E1 27437.062,E2 27437.062} C_VEL
LIN {X 0,Y 576.122,Z 355.032,A -85,B 0,C 180,E1 27434.085,E2 27434.085} C_VEL
LIN {X 0,Y 576.082,Z 355.033,A -85,B 0,C 180,E1 27430.956,E2 27430.956} C_VEL
LIN {X 0,Y 576.142,Z 355.032,A -85,B 0,C 180,E1 27427.877,E2 27427.877} C_VEL
LIN {X 0,Y 576.077,Z 355.033,A -85,B 0,C 180,E1 27424.725,E2 27424.725} C_VEL
LIN {X 0,Y 576.156,Z 355.034,A -85,B 0,C 180,E1 27421.608,E2 27421.608} C_VEL
LIN {X 0,Y 576.078,Z 355.033,A -85,B 0,C 180,E1 27418.505,E2 27418.505} C_VEL
LIN {X 0,Y 576.123,Z 355.034,A -85,B 0,C 180,E1 27415.302,E2 27415.302} C_VEL
LIN {X 0,Y 576.08,Z 355.034,A -85,B 0,C 180,E1 27412.321,E2 27412.321} C_VEL
LIN {X 0,Y 576.099,Z 355.033,A -85,B 0,C 180,E1 27409.023,E2 27409.023} C_VEL
LIN {X 0,Y 576.09,Z 355.033,A -85,B 0,C 180,E1 27406.077,E2 27406.077} C_VEL
LIN {X 0,Y 576.083,Z 355.034,A -85,B 0,C 180,E1 27402.737,E2 27402.737} C_VEL
LIN {X 0,Y 576.107,Z 355.033,A -85,B 0,C 180,E1 27399.823,E2 27399.823} C_VEL
LIN {X 0,Y 576.082,Z 355.034,A -85,B 0,C 180,E1 27396.659,E2 27396.659} C_VEL
LIN {X 0,Y 576.109,Z 355.034,A -85,B 0,C 180,E1 27393.737,E2 27393.737} C_VEL
LIN {X 0,Y 576.08,Z 355.035,A -85,B 0,C 180,E1 27390.567,E2 27390.567} C_VEL
LIN {X 0,Y 576.117,Z 355.032,A -85,B 0,C 180,E1 27387.606,E2 27387.606} C_VEL
LIN {X 0,Y 576.146,Z 355.124,A -85,B 0,C 180,E1 27387.464,E2 27387.464} C_VEL
LIN {X 0,Y 577.421,Z 361.431,A -85,B 0,C 180,E1 27386.683,E2 27386.683} C_VEL
LIN {X 0,Y 577.122,Z 390.031,A -85,B 0,C 180,E1 27383.483,E2 27383.483} C_VEL
LIN {X 0,Y 576.849,Z 419.248,A -85,B 0,C 180,E1 27380.283,E2 27380.283} C_VEL
LIN {X 0,Y 576.566,Z 450.452,A -85,B 0,C 180,E1 27376.938,E2 27376.938} C_VEL
LIN {X 0,Y 576.356,Z 480.964,A -85,B 0,C 180,E1 27373.738,E2 27373.738} C_VEL
LIN {X 0,Y 576.764,Z 488.092,A -85,B 0,C 180,E1 27373.638,E2 27373.638} C_VEL
LIN {X 0,Y 576.547,Z 592.36,A -85,B 0,C 180,E1 27372.311,E2 27372.311} C_VEL
LIN {X 0,Y 576.491,Z 607.967,A -85,B 0,C 180,E1 27371.911,E2 27371.911} C_VEL
LIN {X 0,Y 576.419,Z 620.892,A -85,B 0,C 180,E1 27371.405,E2 27371.405} C_VEL
LIN {X 0,Y 576.297,Z 633.516,A -85,B 0,C 180,E1 27370.749,E2 27370.749} C_VEL
LIN {X 0,Y 576.192,Z 646.658,A -85,B 0,C 180,E1 27369.842,E2 27369.842} C_VEL
LIN {X 0,Y 576.113,Z 657.501,A -85,B 0,C 180,E1 27368.886,E2 27368.886} C_VEL
LIN {X 0,Y 576.029,Z 668.229,A -85,B 0,C 180,E1 27367.681,E2 27367.681} C_VEL
LIN {X 0,Y 575.974,Z 676.536,A -85,B 0,C 180,E1 27366.479,E2 27366.479} C_VEL
LIN {X 0,Y 575.942,Z 683.5,A -85,B 0,C 180,E1 27365.18,E2 27365.18} C_VEL
LIN {X 0,Y 575.922,Z 688.925,A -85,B 0,C 180,E1 27363.783,E2 27363.783} C_VEL
LIN {X 0,Y 575.917,Z 692.561,A -85,B 0,C 180,E1 27362.388,E2 27362.388} C_VEL
LIN {X 0,Y 575.916,Z 694.626,A -85,B 0,C 180,E1 27360.895,E2 27360.895} C_VEL
LIN {X 0,Y 575.915,Z 694.837,A -85,B 0,C 180,E1 27359.403,E2 27359.403} C_VEL
LIN {X 0,Y 575.918,Z 693.292,A -85,B 0,C 180,E1 27357.911,E2 27357.911} C_VEL
LIN {X 0,Y 575.923,Z 690.117,A -85,B 0,C 180,E1 27356.516,E2 27356.516} C_VEL
LIN {X 0,Y 575.933,Z 685.185,A -85,B 0,C 180,E1 27355.12,E2 27355.12} C_VEL
LIN {X 0,Y 575.965,Z 678.287,A -85,B 0,C 180,E1 27353.721,E2 27353.721} C_VEL
LIN {X 0,Y 576.012,Z 670.412,A -85,B 0,C 180,E1 27352.52,E2 27352.52} C_VEL
LIN {X 0,Y 576.083,Z 661.303,A -85,B 0,C 180,E1 27351.416,E2 27351.416} C_VEL
LIN {X 0,Y 576.182,Z 649.641,A -85,B 0,C 180,E1 27350.31,E2 27350.31} C_VEL
LIN {X 0,Y 576.256,Z 638.106,A -85,B 0,C 180,E1 27349.452,E2 27349.452} C_VEL
LIN {X 0,Y 576.397,Z 625.022,A -85,B 0,C 180,E1 27348.696,E2 27348.696} C_VEL
LIN {X 0,Y 576.489,Z 611.267,A -85,B 0,C 180,E1 27348.114,E2 27348.114} C_VEL
LIN {X 0,Y 576.578,Z 596.819,A -85,B 0,C 180,E1 27347.691,E2 27347.691} C_VEL
LIN {X 0,Y 576.619,Z 578.383,A -85,B 0,C 180,E1 27347.399,E2 27347.399} C_VEL
LIN {X 0,Y 576.544,Z 482.244,A -85,B 0,C 180,E1 27346.193,E2 27346.193} C_VEL
LIN {X 0,Y 576.349,Z 480.566,A -85,B 0,C 180,E1 27346.149,E2 27346.149} C_VEL
LIN {X 0,Y 576.564,Z 449.304,A -85,B 0,C 180,E1 27342.849,E2 27342.849} C_VEL
LIN {X 0,Y 576.847,Z 418.434,A -85,B 0,C 180,E1 27339.538,E2 27339.538} C_VEL
LIN {X 0,Y 577.174,Z 388.978,A -85,B 0,C 180,E1 27336.303,E2 27336.303} C_VEL
LIN {X 0,Y 577.585,Z 361.267,A -85,B 0,C 180,E1 27333.14,E2 27333.14} C_VEL
LIN {X 0,Y 576.111,Z 355.038,A -85,B 0,C 180,E1 27332.282,E2 27332.282} C_VEL
LIN {X 0,Y 576.086,Z 355.036,A -85,B 0,C 180,E1 27329.318,E2 27329.318} C_VEL
LIN {X 0,Y 576.086,Z 355.035,A -85,B 0,C 180,E1 27325.903,E2 27325.903} C_VEL
LIN {X 0,Y 576.107,Z 355.034,A -85,B 0,C 180,E1 27322.97,E2 27322.97} C_VEL
LIN {X 0,Y 576.084,Z 355.034,A -85,B 0,C 180,E1 27319.786,E2 27319.786} C_VEL
LIN {X 0,Y 576.13,Z 355.033,A -85,B 0,C 180,E1 27316.724,E2 27316.724} C_VEL
LIN {X 0,Y 576.08,Z 355.034,A -85,B 0,C 180,E1 27313.555,E2 27313.555} C_VEL
LIN {X 0,Y 576.16,Z 355.033,A -85,B 0,C 180,E1 27310.374,E2 27310.374} C_VEL
LIN {X 0,Y 576.08,Z 355.034,A -85,B 0,C 180,E1 27307.282,E2 27307.282} C_VEL
LIN {X 0,Y 576.133,Z 355.036,A -85,B 0,C 180,E1 27304.094,E2 27304.094} C_VEL
LIN {X 0,Y 576.096,Z 355.145,A -85,B 0,C 180,E1 27301.261,E2 27301.261} C_VEL
LIN {X 0,Y 578.812,Z 363.333,A -85,B 0,C 180,E1 27300.522,E2 27300.522} C_VEL
LIN {X 0,Y 578.367,Z 404.357,A -85,B 0,C 180,E1 27297.601,E2 27297.601} C_VEL
LIN {X 0,Y 577.84,Z 450.04,A -85,B 0,C 180,E1 27294.428,E2 27294.428} C_VEL
LIN {X 0,Y 577.795,Z 463.162,A -85,B 0,C 180,E1 27293.555,E2 27293.555} C_VEL
LIN {X 0,Y 578.389,Z 469.397,A -85,B 0,C 180,E1 27293.447,E2 27293.447} C_VEL
LIN {X 0,Y 577.842,Z 672.313,A -85,B 0,C 180,E1 27290.776,E2 27290.776} C_VEL
LIN {X 0,Y 577.693,Z 691.304,A -85,B 0,C 180,E1 27290.336,E2 27290.336} C_VEL
LIN {X 0,Y 577.498,Z 709.397,A -85,B 0,C 180,E1 27289.732,E2 27289.732} C_VEL
LIN {X 0,Y 577.27,Z 727.337,A -85,B 0,C 180,E1 27288.936,E2 27288.936} C_VEL
LIN {X 0,Y 577.028,Z 744.587,A -85,B 0,C 180,E1 27287.965,E2 27287.965} C_VEL
LIN {X 0,Y 576.782,Z 760.967,A -85,B 0,C 180,E1 27286.828,E2 27286.828} C_VEL
LIN {X 0,Y 576.551,Z 776.222,A -85,B 0,C 180,E1 27285.542,E2 27285.542} C_VEL
LIN {X 0,Y 576.349,Z 790.168,A -85,B 0,C 180,E1 27284.126,E2 27284.126} C_VEL
LIN {X 0,Y 576.197,Z 802.458,A -85,B 0,C 180,E1 27282.63,E2 27282.63} C_VEL
LIN {X 0,Y 576.083,Z 813.503,A -85,B 0,C 180,E1 27281.006,E2 27281.006} C_VEL
LIN {X 0,Y 576.007,Z 823.024,A -85,B 0,C 180,E1 27279.29,E2 27279.29} C_VEL
LIN {X 0,Y 575.957,Z 830.583,A -85,B 0,C 180,E1 27277.582,E2 27277.582} C_VEL
LIN {X 0,Y 575.921,Z 836.714,A -85,B 0,C 180,E1 27275.779,E2 27275.779} C_VEL
LIN {X 0,Y 575.918,Z 841.079,A -85,B 0,C 180,E1 27273.982,E2 27273.982} C_VEL
LIN {X 0,Y 575.911,Z 843.901,A -85,B 0,C 180,E1 27272.089,E2 27272.089} C_VEL
LIN {X 0,Y 575.909,Z 844.962,A -85,B 0,C 180,E1 27270.199,E2 27270.199} C_VEL
LIN {X 0,Y 575.91,Z 844.281,A -85,B 0,C 180,E1 27268.309,E2 27268.309} C_VEL
LIN {X 0,Y 575.91,Z 841.846,A -85,B 0,C 180,E1 27266.417,E2 27266.417} C_VEL
LIN {X 0,Y 575.923,Z 837.589,A -85,B 0,C 180,E1 27264.521,E2 27264.521} C_VEL
LIN {X 0,Y 575.952,Z 831.391,A -85,B 0,C 180,E1 27262.619,E2 27262.619} C_VEL
LIN {X 0,Y 576.004,Z 823.538,A -85,B 0,C 180,E1 27260.811,E2 27260.811} C_VEL
LIN {X 0,Y 576.076,Z 814.138,A -85,B 0,C 180,E1 27259.095,E2 27259.095} C_VEL
LIN {X 0,Y 576.192,Z 803.228,A -85,B 0,C 180,E1 27257.472,E2 27257.472} C_VEL
LIN {X 0,Y 576.345,Z 790.798,A -85,B 0,C 180,E1 27255.944,E2 27255.944} C_VEL
LIN {X 0,Y 576.542,Z 776.774,A -85,B 0,C 180,E1 27254.51,E2 27254.51} C_VEL
LIN {X 0,Y 576.769,Z 761.634,A -85,B 0,C 180,E1 27253.224,E2 27253.224} C_VEL
LIN {X 0,Y 577.013,Z 745.399,A -85,B 0,C 180,E1 27252.087,E2 27252.087} C_VEL
LIN {X 0,Y 577.236,Z 729.056,A -85,B 0,C 180,E1 27251.153,E2 27251.153} C_VEL
LIN {X 0,Y 577.454,Z 711.969,A -85,B 0,C 180,E1 27250.372,E2 27250.372} C_VEL
LIN {X 0,Y 577.658,Z 693.471,A -85,B 0,C 180,E1 27249.728,E2 27249.728} C_VEL
LIN {X 0,Y 577.813,Z 674.748,A -85,B 0,C 180,E1 27249.272,E2 27249.272} C_VEL
LIN {X 0,Y 577.93,Z 645.777,A -85,B 0,C 180,E1 27248.854,E2 27248.854} C_VEL
LIN {X 0,Y 578.217,Z 465.841,A -85,B 0,C 180,E1 27246.498,E2 27246.498} C_VEL
LIN {X 0,Y 577.726,Z 462.249,A -85,B 0,C 180,E1 27246.408,E2 27246.408} C_VEL
LIN {X 0,Y 578.222,Z 416.172,A -85,B 0,C 180,E1 27243.227,E2 27243.227} C_VEL
LIN {X 0,Y 578.713,Z 373.639,A -85,B 0,C 180,E1 27240.216,E2 27240.216} C_VEL
LIN {X 0,Y 578.694,Z 362.666,A -85,B 0,C 180,E1 27239.43,E2 27239.43} C_VEL
LIN {X 0,Y 576.079,Z 355.02,A -85,B 0,C 180,E1 27238.709,E2 27238.709} C_VEL
LIN {X 0,Y 576.145,Z 355.033,A -85,B 0,C 180,E1 27235.545,E2 27235.545} C_VEL
LIN {X 0,Y 576.081,Z 355.034,A -85,B 0,C 180,E1 27232.468,E2 27232.468} C_VEL
LIN {X 0,Y 576.12,Z 355.033,A -85,B 0,C 180,E1 27229.266,E2 27229.266} C_VEL
LIN {X 0,Y 576.087,Z 355.034,A -85,B 0,C 180,E1 27226.221,E2 27226.221} C_VEL
LIN {X 0,Y 576.089,Z 355.033,A -85,B 0,C 180,E1 27222.871,E2 27222.871} C_VEL
LIN {X 0,Y 576.101,Z 355.034,A -85,B 0,C 180,E1 27219.953,E2 27219.953} C_VEL
LIN {X 0,Y 576.081,Z 355.034,A -85,B 0,C 180,E1 27216.659,E2 27216.659} C_VEL
LIN {X 0,Y 576.131,Z 355.035,A -85,B 0,C 180,E1 27213.615,E2 27213.615} C_VEL
LIN {X 0,Y 576.076,Z 355.037,A -85,B 0,C 180,E1 27210.451,E2 27210.451} C_VEL
LIN {X 0,Y 576.126,Z 355.263,A -85,B 0,C 180,E1 27207.858,E2 27207.858} C_VEL
LIN {X 0,Y 577.888,Z 361.856,A -85,B 0,C 180,E1 27207.179,E2 27207.179} C_VEL
LIN {X 0,Y 577.55,Z 397.031,A -85,B 0,C 180,E1 27204.115,E2 27204.115} C_VEL
LIN {X 0,Y 577.546,Z 404.519,A -85,B 0,C 180,E1 27203.503,E2 27203.503} C_VEL
LIN {X 0,Y 578.359,Z 410.484,A -85,B 0,C 180,E1 27203.389,E2 27203.389} C_VEL
LIN {X 0,Y 577.842,Z 612.441,A -85,B 0,C 180,E1 27200.73,E2 27200.73} C_VEL
LIN {X 0,Y 577.681,Z 631.849,A -85,B 0,C 180,E1 27200.276,E2 27200.276} C_VEL
LIN {X 0,Y 577.495,Z 649.614,A -85,B 0,C 180,E1 27199.679,E2 27199.679} C_VEL
LIN {X 0,Y 577.256,Z 668.244,A -85,B 0,C 180,E1 27198.846,E2 27198.846} C_VEL
LIN {X 0,Y 577.013,Z 685.537,A -85,B 0,C 180,E1 27197.861,E2 27197.861} C_VEL
LIN {X 0,Y 576.769,Z 701.742,A -85,B 0,C 180,E1 27196.724,E2 27196.724} C_VEL
LIN {X 0,Y 576.537,Z 716.824,A -85,B 0,C 180,E1 27195.439,E2 27195.439} C_VEL
LIN {X 0,Y 576.352,Z 730.417,A -85,B 0,C 180,E1 27194.056,E2 27194.056} C_VEL
LIN {X 0,Y 576.195,Z 742.904,A -85,B 0,C 180,E1 27192.527,E2 27192.527} C_VEL
LIN {X 0,Y 576.079,Z 753.848,A -85,B 0,C 180,E1 27190.905,E2 27190.905} C_VEL
LIN {X 0,Y 576.001,Z 763.306,A -85,B 0,C 180,E1 27189.189,E2 27189.189} C_VEL
LIN {X 0,Y 575.953,Z 771.217,A -85,B 0,C 180,E1 27187.381,E2 27187.381} C_VEL
LIN {X 0,Y 575.928,Z 777.473,A -85,B 0,C 180,E1 27185.479,E2 27185.479} C_VEL
LIN {X 0,Y 575.919,Z 781.769,A -85,B 0,C 180,E1 27183.583,E2 27183.583} C_VEL
LIN {X 0,Y 575.911,Z 784.24,A -85,B 0,C 180,E1 27181.691,E2 27181.691} C_VEL
LIN {X 0,Y 575.916,Z 784.972,A -85,B 0,C 180,E1 27179.801,E2 27179.801} C_VEL
LIN {X 0,Y 575.906,Z 783.964,A -85,B 0,C 180,E1 27177.91,E2 27177.91} C_VEL
LIN {X 0,Y 575.916,Z 781.178,A -85,B 0,C 180,E1 27176.018,E2 27176.018} C_VEL
LIN {X 0,Y 575.921,Z 776.544,A -85,B 0,C 180,E1 27174.121,E2 27174.121} C_VEL
LIN {X 0,Y 575.956,Z 770.374,A -85,B 0,C 180,E1 27172.318,E2 27172.318} C_VEL
LIN {X 0,Y 576,Z 762.754,A -85,B 0,C 180,E1 27170.609,E2 27170.609} C_VEL
LIN {X 0,Y 576.085,Z 753.139,A -85,B 0,C 180,E1 27168.892,E2 27168.892} C_VEL
LIN {X 0,Y 576.203,Z 742.039,A -85,B 0,C 180,E1 27167.269,E2 27167.269} C_VEL
LIN {X 0,Y 576.364,Z 729.374,A -85,B 0,C 180,E1 27165.739,E2 27165.739} C_VEL
LIN {X 0,Y 576.491,Z 721.126,A -85,B 0,C 180,E1 27164.879,E2 27164.879} C_VEL
LIN {X 0,Y 575.605,Z 715.751,A -85,B 0,C 180,E1 27164.327,E2 27164.327} C_VEL
LIN {X 0,Y 569.974,Z 701.875,A -85,B 0,C 180,E1 27162.981,E2 27162.981} C_VEL
LIN {X 0,Y 569.12,Z 695.813,A -85,B 0,C 180,E1 27162.501,E2 27162.501} C_VEL
LIN {X 0,Y 569.415,Z 679.316,A -85,B 0,C 180,E1 27161.415,E2 27161.415} C_VEL
LIN {X 0,Y 569.724,Z 661.951,A -85,B 0,C 180,E1 27160.491,E2 27160.491} C_VEL
LIN {X 0,Y 570.006,Z 643.503,A -85,B 0,C 180,E1 27159.73,E2 27159.73} C_VEL
LIN {X 0,Y 570.229,Z 624.795,A -85,B 0,C 180,E1 27159.164,E2 27159.164} C_VEL
LIN {X 0,Y 570.397,Z 605.186,A -85,B 0,C 180,E1 27158.776,E2 27158.776} C_VEL
LIN {X 0,Y 570.882,Z 409.273,A -85,B 0,C 180,E1 27156.179,E2 27156.179} C_VEL
LIN {X 0,Y 569.902,Z 403.667,A -85,B 0,C 180,E1 27156.032,E2 27156.032} C_VEL
LIN {X 0,Y 570.377,Z 367.26,A -85,B 0,C 180,E1 27152.829,E2 27152.829} C_VEL
LIN {X 0,Y 570.179,Z 362.859,A -85,B 0,C 180,E1 27152.422,E2 27152.422} C_VEL
LIN {X 0,Y 568.145,Z 356.026,A -85,B 0,C 180,E1 27151.687,E2 27151.687} C_VEL
LIN {X 0,Y 568.212,Z 356.023,A -85,B 0,C 180,E1 27148.492,E2 27148.492} C_VEL
LIN {X 0,Y 568.146,Z 356.022,A -85,B 0,C 180,E1 27145.359,E2 27145.359} C_VEL
LIN {X 0,Y 568.166,Z 356.023,A -85,B 0,C 180,E1 27142.036,E2 27142.036} C_VEL
LIN {X 0,Y 568.156,Z 356.021,A -85,B 0,C 180,E1 27139.106,E2 27139.106} C_VEL
LIN {X 0,Y 568.151,Z 356.022,A -85,B 0,C 180,E1 27135.747,E2 27135.747} C_VEL
LIN {X 0,Y 568.196,Z 356.021,A -85,B 0,C 180,E1 27132.648,E2 27132.648} C_VEL
LIN {X 0,Y 568.142,Z 356.022,A -85,B 0,C 180,E1 27129.444,E2 27129.444} C_VEL
LIN {X 0,Y 568.213,Z 356.023,A -85,B 0,C 180,E1 27126.3,E2 27126.3} C_VEL
LIN {X 0,Y 568.143,Z 356.022,A -85,B 0,C 180,E1 27123.184,E2 27123.184} C_VEL
LIN {X 0,Y 568.184,Z 356.022,A -85,B 0,C 180,E1 27119.985,E2 27119.985} C_VEL
LIN {X 0,Y 568.147,Z 356.021,A -85,B 0,C 180,E1 27117.004,E2 27117.004} C_VEL
LIN {X 0,Y 568.158,Z 356.022,A -85,B 0,C 180,E1 27113.656,E2 27113.656} C_VEL
LIN {X 0,Y 568.161,Z 356.021,A -85,B 0,C 180,E1 27110.715,E2 27110.715} C_VEL
LIN {X 0,Y 568.147,Z 356.021,A -85,B 0,C 180,E1 27107.408,E2 27107.408} C_VEL
LIN {X 0,Y 568.189,Z 356.021,A -85,B 0,C 180,E1 27104.366,E2 27104.366} C_VEL
LIN {X 0,Y 568.142,Z 356.022,A -85,B 0,C 180,E1 27101.162,E2 27101.162} C_VEL
LIN {X 0,Y 568.215,Z 356.022,A -85,B 0,C 180,E1 27097.991,E2 27097.991} C_VEL
LIN {X 0,Y 568.143,Z 356.021,A -85,B 0,C 180,E1 27094.846,E2 27094.846} C_VEL
LIN {X 0,Y 568.173,Z 356.022,A -85,B 0,C 180,E1 27091.613,E2 27091.613} C_VEL
LIN {X 0,Y 568.145,Z 356.02,A -85,B 0,C 180,E1 27088.689,E2 27088.689} C_VEL
LIN {X 0,Y 568.157,Z 356.022,A -85,B 0,C 180,E1 27085.357,E2 27085.357} C_VEL
LIN {X 0,Y 568.158,Z 356.02,A -85,B 0,C 180,E1 27082.416,E2 27082.416} C_VEL
LIN {X 0,Y 568.146,Z 356.022,A -85,B 0,C 180,E1 27079.115,E2 27079.115} C_VEL
LIN {X 0,Y 568.19,Z 356.021,A -85,B 0,C 180,E1 27076.049,E2 27076.049} C_VEL
LIN {X 0,Y 568.14,Z 356.021,A -85,B 0,C 180,E1 27072.866,E2 27072.866} C_VEL
LIN {X 0,Y 568.215,Z 356.022,A -85,B 0,C 180,E1 27069.701,E2 27069.701} C_VEL
LIN {X 0,Y 568.139,Z 356.022,A -85,B 0,C 180,E1 27066.673,E2 27066.673} C_VEL
LIN {X 0,Y 568.191,Z 356.022,A -85,B 0,C 180,E1 27063.45,E2 27063.45} C_VEL
LIN {X 0,Y 568.141,Z 356.021,A -85,B 0,C 180,E1 27060.477,E2 27060.477} C_VEL
LIN {X 0,Y 568.175,Z 356.023,A -85,B 0,C 180,E1 27057.264,E2 27057.264} C_VEL
LIN {X 0,Y 568.148,Z 356.023,A -85,B 0,C 180,E1 27054.223,E2 27054.223} C_VEL
LIN {X 0,Y 568.145,Z 356.023,A -85,B 0,C 180,E1 27050.817,E2 27050.817} C_VEL
LIN {X 0,Y 568.186,Z 356.021,A -85,B 0,C 180,E1 27047.761,E2 27047.761} C_VEL
LIN {X 0,Y 568.139,Z 356.022,A -85,B 0,C 180,E1 27044.54,E2 27044.54} C_VEL
LIN {X 0,Y 568.218,Z 356.022,A -85,B 0,C 180,E1 27041.424,E2 27041.424} C_VEL
LIN {X 0,Y 568.138,Z 356.023,A -85,B 0,C 180,E1 27038.287,E2 27038.287} C_VEL
LIN {X 0,Y 568.182,Z 356.024,A -85,B 0,C 180,E1 27035.086,E2 27035.086} C_VEL
LIN {X 0,Y 568.142,Z 356.024,A -85,B 0,C 180,E1 27032.106,E2 27032.106} C_VEL
LIN {X 0,Y 568.159,Z 356.026,A -85,B 0,C 180,E1 27028.789,E2 27028.789} C_VEL
LIN {X 0,Y 568.172,Z 356.104,A -85,B 0,C 180,E1 27027.768,E2 27027.768} C_VEL
LIN {X 0,Y 569.829,Z 363.724,A -85,B 0,C 180,E1 27026.805,E2 27026.805} C_VEL
LIN {X 0,Y 569.449,Z 392.324,A -85,B 0,C 180,E1 27023.573,E2 27023.573} C_VEL
LIN {X 0,Y 569.085,Z 421.204,A -85,B 0,C 180,E1 27020.358,E2 27020.358} C_VEL
LIN {X 0,Y 568.728,Z 452.408,A -85,B 0,C 180,E1 27016.968,E2 27016.968} C_VEL
LIN {X 0,Y 568.48,Z 481.047,A -85,B 0,C 180,E1 27013.932,E2 27013.932} C_VEL
LIN {X 0,Y 568.992,Z 487.762,A -85,B 0,C 180,E1 27013.833,E2 27013.833} C_VEL
LIN {X 0,Y 568.726,Z 592.116,A -85,B 0,C 180,E1 27012.487,E2 27012.487} C_VEL
LIN {X 0,Y 568.662,Z 607.164,A -85,B 0,C 180,E1 27012.106,E2 27012.106} C_VEL
LIN {X 0,Y 568.568,Z 619.799,A -85,B 0,C 180,E1 27011.615,E2 27011.615} C_VEL
LIN {X 0,Y 568.419,Z 632.626,A -85,B 0,C 180,E1 27010.951,E2 27010.951} C_VEL
LIN {X 0,Y 568.272,Z 646.027,A -85,B 0,C 180,E1 27010.032,E2 27010.032} C_VEL
LIN {X 0,Y 568.174,Z 656.969,A -85,B 0,C 180,E1 27009.062,E2 27009.062} C_VEL
LIN {X 0,Y 568.07,Z 667.461,A -85,B 0,C 180,E1 27007.891,E2 27007.891} C_VEL
LIN {X 0,Y 567.994,Z 675.911,A -85,B 0,C 180,E1 27006.672,E2 27006.672} C_VEL
LIN {X 0,Y 567.952,Z 683.043,A -85,B 0,C 180,E1 27005.354,E2 27005.354} C_VEL
LIN {X 0,Y 567.926,Z 688.612,A -85,B 0,C 180,E1 27003.937,E2 27003.937} C_VEL
LIN {X 0,Y 567.919,Z 692.346,A -85,B 0,C 180,E1 27002.523,E2 27002.523} C_VEL
LIN {X 0,Y 567.917,Z 694.561,A -85,B 0,C 180,E1 27001.009,E2 27001.009} C_VEL
LIN {X 0,Y 567.917,Z 694.871,A -85,B 0,C 180,E1 26999.496,E2 26999.496} C_VEL
LIN {X 0,Y 567.916,Z 693.597,A -85,B 0,C 180,E1 26998.083,E2 26998.083} C_VEL
LIN {X 0,Y 567.924,Z 690.412,A -85,B 0,C 180,E1 26996.568,E2 26996.568} C_VEL
LIN {X 0,Y 567.936,Z 685.67,A -85,B 0,C 180,E1 26995.175,E2 26995.175} C_VEL
LIN {X 0,Y 567.972,Z 679.424,A -85,B 0,C 180,E1 26993.836,E2 26993.836} C_VEL
LIN {X 0,Y 568.034,Z 671.138,A -85,B 0,C 180,E1 26992.516,E2 26992.516} C_VEL
LIN {X 0,Y 568.119,Z 662.194,A -85,B 0,C 180,E1 26991.397,E2 26991.397} C_VEL
LIN {X 0,Y 568.245,Z 650.839,A -85,B 0,C 180,E1 26990.275,E2 26990.275} C_VEL
LIN {X 0,Y 568.339,Z 639.571,A -85,B 0,C 180,E1 26989.406,E2 26989.406} C_VEL
LIN {X 0,Y 568.504,Z 626.989,A -85,B 0,C 180,E1 26988.64,E2 26988.64} C_VEL
LIN {X 0,Y 568.636,Z 612.657,A -85,B 0,C 180,E1 26987.999,E2 26987.999} C_VEL
LIN {X 0,Y 568.738,Z 599.161,A -85,B 0,C 180,E1 26987.58,E2 26987.58} C_VEL
LIN {X 0,Y 568.803,Z 583.677,A -85,B 0,C 180,E1 26987.291,E2 26987.291} C_VEL
LIN {X 0,Y 568.77,Z 483.049,A -85,B 0,C 180,E1 26986.011,E2 26986.011} C_VEL
LIN {X 0,Y 568.471,Z 480.56,A -85,B 0,C 180,E1 26985.953,E2 26985.953} C_VEL
LIN {X 0,Y 568.75,Z 449.342,A -85,B 0,C 180,E1 26982.611,E2 26982.611} C_VEL
LIN {X 0,Y 569.096,Z 418.61,A -85,B 0,C 180,E1 26979.267,E2 26979.267} C_VEL
LIN {X 0,Y 569.64,Z 389.483,A -85,B 0,C 180,E1 26975.97,E2 26975.97} C_VEL
LIN {X 0,Y 570.113,Z 363.458,A -85,B 0,C 180,E1 26972.956,E2 26972.956} C_VEL
LIN {X 0,Y 568.146,Z 356.027,A -85,B 0,C 180,E1 26971.945,E2 26971.945} C_VEL
LIN {X 0,Y 568.192,Z 356.024,A -85,B 0,C 180,E1 26968.845,E2 26968.845} C_VEL
LIN {X 0,Y 568.139,Z 356.024,A -85,B 0,C 180,E1 26965.628,E2 26965.628} C_VEL
LIN {X 0,Y 568.211,Z 356.023,A -85,B 0,C 180,E1 26962.494,E2 26962.494} C_VEL
LIN {X 0,Y 568.139,Z 356.024,A -85,B 0,C 180,E1 26959.488,E2 26959.488} C_VEL
LIN {X 0,Y 568.202,Z 356.024,A -85,B 0,C 180,E1 26956.322,E2 26956.322} C_VEL
LIN {X 0,Y 568.145,Z 356.023,A -85,B 0,C 180,E1 26953.204,E2 26953.204} C_VEL
LIN {X 0,Y 568.158,Z 356.024,A -85,B 0,C 180,E1 26949.835,E2 26949.835} C_VEL
LIN {X 0,Y 568.163,Z 356.023,A -85,B 0,C 180,E1 26946.877,E2 26946.877} C_VEL
LIN {X 0,Y 568.146,Z 356.026,A -85,B 0,C 180,E1 26943.546,E2 26943.546} C_VEL
LIN {X 0,Y 568.187,Z 356.275,A -85,B 0,C 180,E1 26941.628,E2 26941.628} C_VEL
LIN {X 0,Y 571.482,Z 366.071,A -85,B 0,C 180,E1 26940.723,E2 26940.723} C_VEL
LIN {X 0,Y 571.006,Z 406.448,A -85,B 0,C 180,E1 26937.837,E2 26937.837} C_VEL
LIN {X 0,Y 570.337,Z 452.403,A -85,B 0,C 180,E1 26934.605,E2 26934.605} C_VEL
LIN {X 0,Y 570.29,Z 463.15,A -85,B 0,C 180,E1 26933.885,E2 26933.885} C_VEL
LIN {X 0,Y 571.047,Z 470.034,A -85,B 0,C 180,E1 26933.758,E2 26933.758} C_VEL
LIN {X 0,Y 570.359,Z 672.313,A -85,B 0,C 180,E1 26931.062,E2 26931.062} C_VEL
LIN {X 0,Y 570.173,Z 691.346,A -85,B 0,C 180,E1 26930.615,E2 26930.615} C_VEL
LIN {X 0,Y 569.929,Z 709.395,A -85,B 0,C 180,E1 26930.005,E2 26930.005} C_VEL
LIN {X 0,Y 569.645,Z 727.108,A -85,B 0,C 180,E1 26929.211,E2 26929.211} C_VEL
LIN {X 0,Y 569.351,Z 743.772,A -85,B 0,C 180,E1 26928.269,E2 26928.269} C_VEL
LIN {X 0,Y 569.055,Z 759.628,A -85,B 0,C 180,E1 26927.169,E2 26927.169} C_VEL
LIN {X 0,Y 568.77,Z 774.557,A -85,B 0,C 180,E1 26925.917,E2 26925.917} C_VEL
LIN {X 0,Y 568.525,Z 788.017,A -85,B 0,C 180,E1 26924.566,E2 26924.566} C_VEL
LIN {X 0,Y 568.308,Z 800.912,A -85,B 0,C 180,E1 26923.015,E2 26923.015} C_VEL
LIN {X 0,Y 568.147,Z 812.229,A -85,B 0,C 180,E1 26921.368,E2 26921.368} C_VEL
LIN {X 0,Y 568.035,Z 821.994,A -85,B 0,C 180,E1 26919.626,E2 26919.626} C_VEL
LIN {X 0,Y 567.965,Z 829.773,A -85,B 0,C 180,E1 26917.892,E2 26917.892} C_VEL
LIN {X 0,Y 567.933,Z 836.111,A -85,B 0,C 180,E1 26916.064,E2 26916.064} C_VEL
LIN {X 0,Y 567.914,Z 840.875,A -85,B 0,C 180,E1 26914.139,E2 26914.139} C_VEL
LIN {X 0,Y 567.911,Z 843.79,A -85,B 0,C 180,E1 26912.22,E2 26912.22} C_VEL
LIN {X 0,Y 567.907,Z 844.94,A -85,B 0,C 180,E1 26910.303,E2 26910.303} C_VEL
LIN {X 0,Y 567.914,Z 844.416,A -85,B 0,C 180,E1 26908.487,E2 26908.487} C_VEL
LIN {X 0,Y 567.909,Z 842.164,A -85,B 0,C 180,E1 26906.568,E2 26906.568} C_VEL
LIN {X 0,Y 567.926,Z 838.351,A -85,B 0,C 180,E1 26904.747,E2 26904.747} C_VEL
LIN {X 0,Y 567.954,Z 832.819,A -85,B 0,C 180,E1 26902.921,E2 26902.921} C_VEL
LIN {X 0,Y 568,Z 825.426,A -85,B 0,C 180,E1 26901.089,E2 26901.089} C_VEL
LIN {X 0,Y 568.093,Z 816.514,A -85,B 0,C 180,E1 26899.35,E2 26899.35} C_VEL
LIN {X 0,Y 568.231,Z 806.149,A -85,B 0,C 180,E1 26897.707,E2 26897.707} C_VEL
LIN {X 0,Y 568.414,Z 794.349,A -85,B 0,C 180,E1 26896.159,E2 26896.159} C_VEL
LIN {X 0,Y 568.647,Z 781.083,A -85,B 0,C 180,E1 26894.707,E2 26894.707} C_VEL
LIN {X 0,Y 568.927,Z 766.225,A -85,B 0,C 180,E1 26893.354,E2 26893.354} C_VEL
LIN {X 0,Y 569.234,Z 750.307,A -85,B 0,C 180,E1 26892.156,E2 26892.156} C_VEL
LIN {X 0,Y 569.54,Z 733.144,A -85,B 0,C 180,E1 26891.106,E2 26891.106} C_VEL
LIN {X 0,Y 569.834,Z 715.803,A -85,B 0,C 180,E1 26890.259,E2 26890.259} C_VEL
LIN {X 0,Y 570.097,Z 697.624,A -85,B 0,C 180,E1 26889.576,E2 26889.576} C_VEL
LIN {X 0,Y 570.3,Z 679.019,A -85,B 0,C 180,E1 26889.075,E2 26889.075} C_VEL
LIN {X 0,Y 570.429,Z 658.857,A -85,B 0,C 180,E1 26888.736,E2 26888.736} C_VEL
LIN {X 0,Y 570.9,Z 467.082,A -85,B 0,C 180,E1 26886.195,E2 26886.195} C_VEL
LIN {X 0,Y 570.225,Z 462.249,A -85,B 0,C 180,E1 26886.078,E2 26886.078} C_VEL
LIN {X 0,Y 570.892,Z 414.596,A -85,B 0,C 180,E1 26882.742,E2 26882.742} C_VEL
LIN {X 0,Y 571.379,Z 373.545,A -85,B 0,C 180,E1 26879.82,E2 26879.82} C_VEL
LIN {X 0,Y 571.35,Z 365.41,A -85,B 0,C 180,E1 26879.232,E2 26879.232} C_VEL
LIN {X 0,Y 568.152,Z 356.008,A -85,B 0,C 180,E1 26878.34,E2 26878.34} C_VEL
LIN {X 0,Y 568.149,Z 356.022,A -85,B 0,C 180,E1 26874.99,E2 26874.99} C_VEL
LIN {X 0,Y 568.177,Z 356.023,A -85,B 0,C 180,E1 26871.981,E2 26871.981} C_VEL
LIN {X 0,Y 568.146,Z 356.022,A -85,B 0,C 180,E1 26868.838,E2 26868.838} C_VEL
LIN {X 0,Y 568.204,Z 356.023,A -85,B 0,C 180,E1 26865.685,E2 26865.685} C_VEL
LIN {X 0,Y 568.139,Z 356.023,A -85,B 0,C 180,E1 26862.49,E2 26862.49} C_VEL
LIN {X 0,Y 568.201,Z 356.023,A -85,B 0,C 180,E1 26859.308,E2 26859.308} C_VEL
LIN {X 0,Y 568.141,Z 356.023,A -85,B 0,C 180,E1 26856.251,E2 26856.251} C_VEL
LIN {X 0,Y 568.177,Z 356.025,A -85,B 0,C 180,E1 26853.061,E2 26853.061} C_VEL
LIN {X 0,Y 568.147,Z 356.027,A -85,B 0,C 180,E1 26850.019,E2 26850.019} C_VEL
LIN {X 0,Y 568.14,Z 356.034,A -85,B 0,C 180,E1 26848.183,E2 26848.183} C_VEL
LIN {X 0,Y 570.412,Z 364.377,A -85,B 0,C 180,E1 26847.339,E2 26847.339} C_VEL
LIN {X 0,Y 569.963,Z 399.552,A -85,B 0,C 180,E1 26844.236,E2 26844.236} C_VEL
LIN {X 0,Y 569.977,Z 404.553,A -85,B 0,C 180,E1 26843.835,E2 26843.835} C_VEL
LIN {X 0,Y 571.015,Z 411.41,A -85,B 0,C 180,E1 26843.696,E2 26843.696} C_VEL
LIN {X 0,Y 570.356,Z 612.479,A -85,B 0,C 180,E1 26841.015,E2 26841.015} C_VEL
LIN {X 0,Y 570.157,Z 631.967,A -85,B 0,C 180,E1 26840.553,E2 26840.553} C_VEL
LIN {X 0,Y 569.925,Z 649.632,A -85,B 0,C 180,E1 26839.951,E2 26839.951} C_VEL
LIN {X 0,Y 569.626,Z 668.266,A -85,B 0,C 180,E1 26839.109,E2 26839.109} C_VEL
LIN {X 0,Y 569.318,Z 685.545,A -85,B 0,C 180,E1 26838.111,E2 26838.111} C_VEL
LIN {X 0,Y 569.011,Z 701.757,A -85,B 0,C 180,E1 26836.959,E2 26836.959} C_VEL
LIN {X 0,Y 568.717,Z 716.829,A -85,B 0,C 180,E1 26835.656,E2 26835.656} C_VEL
LIN {X 0,Y 568.48,Z 730.427,A -85,B 0,C 180,E1 26834.255,E2 26834.255} C_VEL
LIN {X 0,Y 568.276,Z 742.913,A -85,B 0,C 180,E1 26832.705,E2 26832.705} C_VEL
LIN {X 0,Y 568.127,Z 753.849,A -85,B 0,C 180,E1 26831.06,E2 26831.06} C_VEL
LIN {X 0,Y 568.027,Z 763.303,A -85,B 0,C 180,E1 26829.319,E2 26829.319} C_VEL
LIN {X 0,Y 567.964,Z 771.215,A -85,B 0,C 180,E1 26827.485,E2 26827.485} C_VEL
LIN {X 0,Y 567.933,Z 777.18,A -85,B 0,C 180,E1 26825.658,E2 26825.658} C_VEL
LIN {X 0,Y 567.918,Z 781.385,A -85,B 0,C 180,E1 26823.836,E2 26823.836} C_VEL
LIN {X 0,Y 567.908,Z 784.074,A -85,B 0,C 180,E1 26821.917,E2 26821.917} C_VEL
LIN {X 0,Y 567.914,Z 784.996,A -85,B 0,C 180,E1 26820,E2 26820} C_VEL
LIN {X 0,Y 567.905,Z 784.146,A -85,B 0,C 180,E1 26818.083,E2 26818.083} C_VEL
LIN {X 0,Y 567.915,Z 781.554,A -85,B 0,C 180,E1 26816.164,E2 26816.164} C_VEL
LIN {X 0,Y 567.924,Z 777.442,A -85,B 0,C 180,E1 26814.342,E2 26814.342} C_VEL
LIN {X 0,Y 567.955,Z 771.535,A -85,B 0,C 180,E1 26812.514,E2 26812.514} C_VEL
LIN {X 0,Y 568.018,Z 763.734,A -85,B 0,C 180,E1 26810.68,E2 26810.68} C_VEL
LIN {X 0,Y 568.125,Z 754.405,A -85,B 0,C 180,E1 26808.94,E2 26808.94} C_VEL
LIN {X 0,Y 568.269,Z 743.583,A -85,B 0,C 180,E1 26807.295,E2 26807.295} C_VEL
LIN {X 0,Y 568.463,Z 731.085,A -85,B 0,C 180,E1 26805.731,E2 26805.731} C_VEL
LIN {X 0,Y 568.708,Z 717.231,A -85,B 0,C 180,E1 26804.291,E2 26804.291} C_VEL
LIN {X 0,Y 568.999,Z 702.219,A -85,B 0,C 180,E1 26802.987,E2 26802.987} C_VEL
LIN {X 0,Y 569.12,Z 695.813,A -85,B 0,C 180,E1 26802.501,E2 26802.501} C_VEL
LIN {X 0,Y 568.291,Z 689.636,A -85,B 0,C 180,E1 26802.035,E2 26802.035} C_VEL
LIN {X 0,Y 562.854,Z 674.02,A -85,B 0,C 180,E1 26800.871,E2 26800.871} C_VEL
LIN {X 0,Y 562.027,Z 667.326,A -85,B 0,C 180,E1 26800.483,E2 26800.483} C_VEL
LIN {X 0,Y 562.386,Z 649.197,A -85,B 0,C 180,E1 26799.661,E2 26799.661} C_VEL
LIN {X 0,Y 562.675,Z 630.308,A -85,B 0,C 180,E1 26799.022,E2 26799.022} C_VEL
LIN {X 0,Y 562.895,Z 611.469,A -85,B 0,C 180,E1 26798.585,E2 26798.585} C_VEL
LIN {X 0,Y 563.571,Z 410.551,A -85,B 0,C 180,E1 26795.869,E2 26795.869} C_VEL
LIN {X 0,Y 562.347,Z 403.71,A -85,B 0,C 180,E1 26795.694,E2 26795.694} C_VEL
LIN {X 0,Y 562.875,Z 368.984,A -85,B 0,C 180,E1 26792.608,E2 26792.608} C_VEL
LIN {X 0,Y 562.598,Z 365.158,A -85,B 0,C 180,E1 26792.249,E2 26792.249} C_VEL
LIN {X 0,Y 560.211,Z 357.016,A -85,B 0,C 180,E1 26791.366,E2 26791.366} C_VEL
LIN {X 0,Y 560.218,Z 357.012,A -85,B 0,C 180,E1 26787.97,E2 26787.97} C_VEL
LIN {X 0,Y 560.239,Z 357.011,A -85,B 0,C 180,E1 26784.923,E2 26784.923} C_VEL
LIN {X 0,Y 560.209,Z 357.012,A -85,B 0,C 180,E1 26781.733,E2 26781.733} C_VEL
LIN {X 0,Y 560.262,Z 357.01,A -85,B 0,C 180,E1 26778.676,E2 26778.676} C_VEL
LIN {X 0,Y 560.203,Z 357.011,A -85,B 0,C 180,E1 26775.458,E2 26775.458} C_VEL
LIN {X 0,Y 560.265,Z 357.012,A -85,B 0,C 180,E1 26772.284,E2 26772.284} C_VEL
LIN {X 0,Y 560.208,Z 357.01,A -85,B 0,C 180,E1 26769.185,E2 26769.185} C_VEL
LIN {X 0,Y 560.224,Z 357.011,A -85,B 0,C 180,E1 26765.831,E2 26765.831} C_VEL
LIN {X 0,Y 560.227,Z 357.01,A -85,B 0,C 180,E1 26762.795,E2 26762.795} C_VEL
LIN {X 0,Y 560.207,Z 357.01,A -85,B 0,C 180,E1 26759.512,E2 26759.512} C_VEL
LIN {X 0,Y 560.267,Z 357.01,A -85,B 0,C 180,E1 26756.378,E2 26756.378} C_VEL
LIN {X 0,Y 560.202,Z 357.01,A -85,B 0,C 180,E1 26753.193,E2 26753.193} C_VEL
LIN {X 0,Y 560.267,Z 357.012,A -85,B 0,C 180,E1 26750.038,E2 26750.038} C_VEL
LIN {X 0,Y 560.208,Z 357.009,A -85,B 0,C 180,E1 26746.913,E2 26746.913} C_VEL
LIN {X 0,Y 560.218,Z 357.01,A -85,B 0,C 180,E1 26743.521,E2 26743.521} C_VEL
LIN {X 0,Y 560.235,Z 357.01,A -85,B 0,C 180,E1 26740.46,E2 26740.46} C_VEL
LIN {X 0,Y 560.203,Z 357.01,A -85,B 0,C 180,E1 26737.177,E2 26737.177} C_VEL
LIN {X 0,Y 560.273,Z 357.01,A -85,B 0,C 180,E1 26733.977,E2 26733.977} C_VEL
LIN {X 0,Y 560.203,Z 357.01,A -85,B 0,C 180,E1 26730.818,E2 26730.818} C_VEL
LIN {X 0,Y 560.246,Z 357.01,A -85,B 0,C 180,E1 26727.647,E2 26727.647} C_VEL
LIN {X 0,Y 560.21,Z 357.01,A -85,B 0,C 180,E1 26724.572,E2 26724.572} C_VEL
LIN {X 0,Y 560.209,Z 357.011,A -85,B 0,C 180,E1 26721.171,E2 26721.171} C_VEL
LIN {X 0,Y 560.253,Z 357.01,A -85,B 0,C 180,E1 26718.052,E2 26718.052} C_VEL
LIN {X 0,Y 560.203,Z 357.011,A -85,B 0,C 180,E1 26714.895,E2 26714.895} C_VEL
LIN {X 0,Y 560.271,Z 357.012,A -85,B 0,C 180,E1 26711.694,E2 26711.694} C_VEL
LIN {X 0,Y 560.205,Z 357.01,A -85,B 0,C 180,E1 26708.538,E2 26708.538} C_VEL
LIN {X 0,Y 560.223,Z 357.011,A -85,B 0,C 180,E1 26705.202,E2 26705.202} C_VEL
LIN {X 0,Y 560.225,Z 357.01,A -85,B 0,C 180,E1 26702.121,E2 26702.121} C_VEL
LIN {X 0,Y 560.204,Z 357.011,A -85,B 0,C 180,E1 26698.829,E2 26698.829} C_VEL
LIN {X 0,Y 560.266,Z 357.012,A -85,B 0,C 180,E1 26695.671,E2 26695.671} C_VEL
LIN {X 0,Y 560.199,Z 357.012,A -85,B 0,C 180,E1 26692.509,E2 26692.509} C_VEL
LIN {X 0,Y 560.256,Z 357.011,A -85,B 0,C 180,E1 26689.33,E2 26689.33} C_VEL
LIN {X 0,Y 560.202,Z 357.011,A -85,B 0,C 180,E1 26686.291,E2 26686.291} C_VEL
LIN {X 0,Y 560.222,Z 357.012,A -85,B 0,C 180,E1 26682.966,E2 26682.966} C_VEL
LIN {X 0,Y 560.216,Z 357.012,A -85,B 0,C 180,E1 26679.98,E2 26679.98} C_VEL
LIN {X 0,Y 560.208,Z 357.012,A -85,B 0,C 180,E1 26676.72,E2 26676.72} C_VEL
LIN {X 0,Y 560.234,Z 357.013,A -85,B 0,C 180,E1 26673.714,E2 26673.714} C_VEL
LIN {X 0,Y 560.2,Z 357.014,A -85,B 0,C 180,E1 26670.449,E2 26670.449} C_VEL
LIN {X 0,Y 560.211,Z 357.08,A -85,B 0,C 180,E1 26668.082,E2 26668.082} C_VEL
LIN {X 0,Y 562.243,Z 365.698,A -85,B 0,C 180,E1 26666.967,E2 26666.967} C_VEL
LIN {X 0,Y 561.763,Z 395.123,A -85,B 0,C 180,E1 26663.608,E2 26663.608} C_VEL
LIN {X 0,Y 561.321,Z 423.727,A -85,B 0,C 180,E1 26660.38,E2 26660.38} C_VEL
LIN {X 0,Y 560.884,Z 454.852,A -85,B 0,C 180,E1 26656.946,E2 26656.946} C_VEL
LIN {X 0,Y 560.604,Z 481.058,A -85,B 0,C 180,E1 26654.132,E2 26654.132} C_VEL
LIN {X 0,Y 561.225,Z 488.194,A -85,B 0,C 180,E1 26654.024,E2 26654.024} C_VEL
LIN {X 0,Y 560.912,Z 591.976,A -85,B 0,C 180,E1 26652.665,E2 26652.665} C_VEL
LIN {X 0,Y 560.828,Z 607.244,A -85,B 0,C 180,E1 26652.275,E2 26652.275} C_VEL
LIN {X 0,Y 560.711,Z 620.062,A -85,B 0,C 180,E1 26651.768,E2 26651.768} C_VEL
LIN {X 0,Y 560.554,Z 631.451,A -85,B 0,C 180,E1 26651.175,E2 26651.175} C_VEL
LIN {X 0,Y 560.386,Z 643.782,A -85,B 0,C 180,E1 26650.354,E2 26650.354} C_VEL
LIN {X 0,Y 560.25,Z 655.387,A -85,B 0,C 180,E1 26649.347,E2 26649.347} C_VEL
LIN {X 0,Y 560.133,Z 664.942,A -85,B 0,C 180,E1 26648.314,E2 26648.314} C_VEL
LIN {X 0,Y 560.028,Z 674.666,A -85,B 0,C 180,E1 26646.973,E2 26646.973} C_VEL
LIN {X 0,Y 559.967,Z 681.525,A -85,B 0,C 180,E1 26645.739,E2 26645.739} C_VEL
LIN {X 0,Y 559.935,Z 687.231,A -85,B 0,C 180,E1 26644.404,E2 26644.404} C_VEL
LIN {X 0,Y 559.92,Z 691.689,A -85,B 0,C 180,E1 26642.866,E2 26642.866} C_VEL
LIN {X 0,Y 559.916,Z 693.988,A -85,B 0,C 180,E1 26641.535,E2 26641.535} C_VEL
LIN {X 0,Y 559.916,Z 694.996,A -85,B 0,C 180,E1 26640,E2 26640} C_VEL
LIN {X 0,Y 559.918,Z 694.102,A -85,B 0,C 180,E1 26638.465,E2 26638.465} C_VEL
LIN {X 0,Y 559.918,Z 691.88,A -85,B 0,C 180,E1 26637.134,E2 26637.134} C_VEL
LIN {X 0,Y 559.932,Z 687.91,A -85,B 0,C 180,E1 26635.699,E2 26635.699} C_VEL
LIN {X 0,Y 559.965,Z 681.969,A -85,B 0,C 180,E1 26634.261,E2 26634.261} C_VEL
LIN {X 0,Y 560.021,Z 675.209,A -85,B 0,C 180,E1 26633.027,E2 26633.027} C_VEL
LIN {X 0,Y 560.117,Z 666.556,A -85,B 0,C 180,E1 26631.79,E2 26631.79} C_VEL
LIN {X 0,Y 560.24,Z 656.301,A -85,B 0,C 180,E1 26630.653,E2 26630.653} C_VEL
LIN {X 0,Y 560.386,Z 645.231,A -85,B 0,C 180,E1 26629.67,E2 26629.67} C_VEL
LIN {X 0,Y 560.546,Z 632.386,A -85,B 0,C 180,E1 26628.789,E2 26628.789} C_VEL
LIN {X 0,Y 560.706,Z 620.581,A -85,B 0,C 180,E1 26628.167,E2 26628.167} C_VEL
LIN {X 0,Y 560.848,Z 607.579,A -85,B 0,C 180,E1 26627.647,E2 26627.647} C_VEL
LIN {X 0,Y 560.957,Z 592.087,A -85,B 0,C 180,E1 26627.248,E2 26627.248} C_VEL
LIN {X 0,Y 561.182,Z 505.641,A -85,B 0,C 180,E1 26626.111,E2 26626.111} C_VEL
LIN {X 0,Y 560.986,Z 483.675,A -85,B 0,C 180,E1 26625.822,E2 26625.822} C_VEL
LIN {X 0,Y 560.597,Z 480.554,A -85,B 0,C 180,E1 26625.751,E2 26625.751} C_VEL
LIN {X 0,Y 560.946,Z 449.335,A -85,B 0,C 180,E1 26622.361,E2 26622.361} C_VEL
LIN {X 0,Y 561.483,Z 419.765,A -85,B 0,C 180,E1 26619.027,E2 26619.027} C_VEL
LIN {X 0,Y 562.139,Z 390.617,A -85,B 0,C 180,E1 26615.685,E2 26615.685} C_VEL
LIN {X 0,Y 562.633,Z 366.116,A -85,B 0,C 180,E1 26612.825,E2 26612.825} C_VEL
LIN {X 0,Y 560.203,Z 357.017,A -85,B 0,C 180,E1 26611.54,E2 26611.54} C_VEL
LIN {X 0,Y 560.247,Z 357.014,A -85,B 0,C 180,E1 26608.352,E2 26608.352} C_VEL
LIN {X 0,Y 560.207,Z 357.013,A -85,B 0,C 180,E1 26605.295,E2 26605.295} C_VEL
LIN {X 0,Y 560.209,Z 357.013,A -85,B 0,C 180,E1 26601.863,E2 26601.863} C_VEL
LIN {X 0,Y 560.237,Z 357.012,A -85,B 0,C 180,E1 26598.864,E2 26598.864} C_VEL
LIN {X 0,Y 560.203,Z 357.013,A -85,B 0,C 180,E1 26595.601,E2 26595.601} C_VEL
LIN {X 0,Y 560.271,Z 357.012,A -85,B 0,C 180,E1 26592.422,E2 26592.422} C_VEL
LIN {X 0,Y 560.202,Z 357.013,A -85,B 0,C 180,E1 26589.317,E2 26589.317} C_VEL
LIN {X 0,Y 560.249,Z 357.013,A -85,B 0,C 180,E1 26586.082,E2 26586.082} C_VEL
LIN {X 0,Y 560.214,Z 357.015,A -85,B 0,C 180,E1 26582.981,E2 26582.981} C_VEL
LIN {X 0,Y 560.273,Z 357.184,A -85,B 0,C 180,E1 26582.04,E2 26582.04} C_VEL
LIN {X 0,Y 564.152,Z 368.766,A -85,B 0,C 180,E1 26580.929,E2 26580.929} C_VEL
LIN {X 0,Y 563.562,Z 410.385,A -85,B 0,C 180,E1 26577.928,E2 26577.928} C_VEL
LIN {X 0,Y 562.827,Z 455.554,A -85,B 0,C 180,E1 26574.732,E2 26574.732} C_VEL
LIN {X 0,Y 562.807,Z 463.168,A -85,B 0,C 180,E1 26574.222,E2 26574.222} C_VEL
LIN {X 0,Y 563.722,Z 471.1,A -85,B 0,C 180,E1 26574.072,E2 26574.072} C_VEL
LIN {X 0,Y 562.892,Z 672.312,A -85,B 0,C 180,E1 26571.355,E2 26571.355} C_VEL
LIN {X 0,Y 562.667,Z 691.314,A -85,B 0,C 180,E1 26570.904,E2 26570.904} C_VEL
LIN {X 0,Y 562.373,Z 709.392,A -85,B 0,C 180,E1 26570.286,E2 26570.286} C_VEL
LIN {X 0,Y 562.029,Z 727.135,A -85,B 0,C 180,E1 26569.48,E2 26569.48} C_VEL
LIN {X 0,Y 561.67,Z 743.768,A -85,B 0,C 180,E1 26568.527,E2 26568.527} C_VEL
LIN {X 0,Y 561.31,Z 759.625,A -85,B 0,C 180,E1 26567.413,E2 26567.413} C_VEL
LIN {X 0,Y 560.954,Z 774.907,A -85,B 0,C 180,E1 26566.111,E2 26566.111} C_VEL
LIN {X 0,Y 560.645,Z 788.943,A -85,B 0,C 180,E1 26564.67,E2 26564.67} C_VEL
LIN {X 0,Y 560.379,Z 802.086,A -85,B 0,C 180,E1 26563.043,E2 26563.043} C_VEL
LIN {X 0,Y 560.193,Z 812.866,A -85,B 0,C 180,E1 26561.427,E2 26561.427} C_VEL
LIN {X 0,Y 560.058,Z 822.508,A -85,B 0,C 180,E1 26559.661,E2 26559.661} C_VEL
LIN {X 0,Y 559.976,Z 830.178,A -85,B 0,C 180,E1 26557.902,E2 26557.902} C_VEL
LIN {X 0,Y 559.936,Z 836.413,A -85,B 0,C 180,E1 26556.048,E2 26556.048} C_VEL
LIN {X 0,Y 559.913,Z 840.876,A -85,B 0,C 180,E1 26554.199,E2 26554.199} C_VEL
LIN {X 0,Y 559.911,Z 843.791,A -85,B 0,C 180,E1 26552.252,E2 26552.252} C_VEL
LIN {X 0,Y 559.908,Z 844.94,A -85,B 0,C 180,E1 26550.307,E2 26550.307} C_VEL
LIN {X 0,Y 559.913,Z 844.416,A -85,B 0,C 180,E1 26548.465,E2 26548.465} C_VEL
LIN {X 0,Y 559.909,Z 842.164,A -85,B 0,C 180,E1 26546.519,E2 26546.519} C_VEL
LIN {X 0,Y 559.929,Z 838.35,A -85,B 0,C 180,E1 26544.672,E2 26544.672} C_VEL
LIN {X 0,Y 559.962,Z 832.818,A -85,B 0,C 180,E1 26542.82,E2 26542.82} C_VEL
LIN {X 0,Y 560.027,Z 825.427,A -85,B 0,C 180,E1 26540.961,E2 26540.961} C_VEL
LIN {X 0,Y 560.136,Z 816.516,A -85,B 0,C 180,E1 26539.197,E2 26539.197} C_VEL
LIN {X 0,Y 560.307,Z 806.151,A -85,B 0,C 180,E1 26537.53,E2 26537.53} C_VEL
LIN {X 0,Y 560.532,Z 794.35,A -85,B 0,C 180,E1 26535.96,E2 26535.96} C_VEL
LIN {X 0,Y 560.823,Z 780.803,A -85,B 0,C 180,E1 26534.46,E2 26534.46} C_VEL
LIN {X 0,Y 561.16,Z 766.032,A -85,B 0,C 180,E1 26533.099,E2 26533.099} C_VEL
LIN {X 0,Y 561.528,Z 750.23,A -85,B 0,C 180,E1 26531.898,E2 26531.898} C_VEL
LIN {X 0,Y 561.9,Z 733.048,A -85,B 0,C 180,E1 26530.834,E2 26530.834} C_VEL
LIN {X 0,Y 562.254,Z 715.805,A -85,B 0,C 180,E1 26529.981,E2 26529.981} C_VEL
LIN {X 0,Y 562.572,Z 697.518,A -85,B 0,C 180,E1 26529.287,E2 26529.287} C_VEL
LIN {X 0,Y 562.819,Z 678.862,A -85,B 0,C 180,E1 26528.78,E2 26528.78} C_VEL
LIN {X 0,Y 562.975,Z 658.603,A -85,B 0,C 180,E1 26528.437,E2 26528.437} C_VEL
LIN {X 0,Y 563.575,Z 468.128,A -85,B 0,C 180,E1 26525.881,E2 26525.881} C_VEL
LIN {X 0,Y 562.737,Z 462.236,A -85,B 0,C 180,E1 26525.739,E2 26525.739} C_VEL
LIN {X 0,Y 563.538,Z 414.493,A -85,B 0,C 180,E1 26522.356,E2 26522.356} C_VEL
LIN {X 0,Y 564.083,Z 371.111,A -85,B 0,C 180,E1 26519.25,E2 26519.25} C_VEL
LIN {X 0,Y 563.974,Z 368.036,A -85,B 0,C 180,E1 26519.012,E2 26519.012} C_VEL
LIN {X 0,Y 560.252,Z 356.997,A -85,B 0,C 180,E1 26517.931,E2 26517.931} C_VEL
LIN {X 0,Y 560.203,Z 357.012,A -85,B 0,C 180,E1 26514.795,E2 26514.795} C_VEL
LIN {X 0,Y 560.278,Z 357.009,A -85,B 0,C 180,E1 26511.576,E2 26511.576} C_VEL
LIN {X 0,Y 560.202,Z 357.012,A -85,B 0,C 180,E1 26508.534,E2 26508.534} C_VEL
LIN {X 0,Y 560.254,Z 357.012,A -85,B 0,C 180,E1 26505.319,E2 26505.319} C_VEL
LIN {X 0,Y 560.208,Z 357.012,A -85,B 0,C 180,E1 26502.209,E2 26502.209} C_VEL
LIN {X 0,Y 560.209,Z 357.012,A -85,B 0,C 180,E1 26498.79,E2 26498.79} C_VEL
LIN {X 0,Y 560.244,Z 357.013,A -85,B 0,C 180,E1 26495.704,E2 26495.704} C_VEL
LIN {X 0,Y 560.201,Z 357.015,A -85,B 0,C 180,E1 26492.495,E2 26492.495} C_VEL
LIN {X 0,Y 560.273,Z 357.012,A -85,B 0,C 180,E1 26489.391,E2 26489.391} C_VEL
LIN {X 0,Y 560.235,Z 357.267,A -85,B 0,C 180,E1 26488.458,E2 26488.458} C_VEL
LIN {X 0,Y 562.856,Z 366.483,A -85,B 0,C 180,E1 26487.507,E2 26487.507} C_VEL
LIN {X 0,Y 562.578,Z 388.991,A -85,B 0,C 180,E1 26485.52,E2 26485.52} C_VEL
LIN {X 0,Y 562.404,Z 404.448,A -85,B 0,C 180,E1 26484.178,E2 26484.178} C_VEL
LIN {X 0,Y 563.687,Z 412.642,A -85,B 0,C 180,E1 26484.007,E2 26484.007} C_VEL
LIN {X 0,Y 562.888,Z 612.515,A -85,B 0,C 180,E1 26481.307,E2 26481.307} C_VEL
LIN {X 0,Y 562.649,Z 632.014,A -85,B 0,C 180,E1 26480.839,E2 26480.839} C_VEL
LIN {X 0,Y 562.369,Z 649.65,A -85,B 0,C 180,E1 26480.231,E2 26480.231} C_VEL
LIN {X 0,Y 562.008,Z 668.283,A -85,B 0,C 180,E1 26479.378,E2 26479.378} C_VEL
LIN {X 0,Y 561.633,Z 685.553,A -85,B 0,C 180,E1 26478.367,E2 26478.367} C_VEL
LIN {X 0,Y 561.262,Z 701.771,A -85,B 0,C 180,E1 26477.201,E2 26477.201} C_VEL
LIN {X 0,Y 560.905,Z 716.833,A -85,B 0,C 180,E1 26475.88,E2 26475.88} C_VEL
LIN {X 0,Y 560.608,Z 730.697,A -85,B 0,C 180,E1 26474.428,E2 26474.428} C_VEL
LIN {X 0,Y 560.365,Z 742.921,A -85,B 0,C 180,E1 26472.887,E2 26472.887} C_VEL
LIN {X 0,Y 560.176,Z 753.85,A -85,B 0,C 180,E1 26471.219,E2 26471.219} C_VEL
LIN {X 0,Y 560.05,Z 763.3,A -85,B 0,C 180,E1 26469.453,E2 26469.453} C_VEL
LIN {X 0,Y 559.977,Z 771.213,A -85,B 0,C 180,E1 26467.593,E2 26467.593} C_VEL
LIN {X 0,Y 559.937,Z 777.182,A -85,B 0,C 180,E1 26465.739,E2 26465.739} C_VEL
LIN {X 0,Y 559.917,Z 781.381,A -85,B 0,C 180,E1 26463.891,E2 26463.891} C_VEL
LIN {X 0,Y 559.909,Z 784.07,A -85,B 0,C 180,E1 26461.944,E2 26461.944} C_VEL
LIN {X 0,Y 559.914,Z 784.996,A -85,B 0,C 180,E1 26460,E2 26460} C_VEL
